LIN {X -0.149,Y -605.682,Z 1425.041,A 0.000,B 0.000,C 90.000,E1 43.299} C_DIS
LIN {X -0.289,Y -605.290,Z 1425.036,A 0.000,B 0.000,C 90.000,E1 42.528} C_DIS
LIN {X -0.379,Y -604.390,Z 1425.029,A 0.000,B 0.000,C 90.000,E1 41.229} C_DIS
LIN {X -0.024,Y -603.135,Z 1425.022,A 0.000,B 0.000,C 90.000,E1 39.886} C_DIS
LIN {X -0.162,Y -601.577,Z 1425.014,A 0.000,B 0.000,C 90.000,E1 38.588} C_DIS
LIN {X 0.234,Y -599.735,Z 1425.007,A 0.000,B 0.000,C 90.000,E1 37.237} C_DIS
LIN {X 0.126,Y -598.447,Z 1425.003,A 0.000,B 0.000,C 90.000,E1 36.457} C_DIS
LIN {X 0.240,Y -596.428,Z 1424.997,A 0.000,B 0.000,C 90.000,E1 35.391} C_DIS
LIN {X 0.320,Y -594.156,Z 1424.991,A 0.000,B 0.000,C 90.000,E1 34.326} C_DIS
LIN {X -0.182,Y -592.218,Z 1424.986,A 0.000,B 0.000,C 90.000,E1 33.579} C_DIS
LIN {X 0.002,Y -589.416,Z 1424.981,A 0.000,B 0.000,C 90.000,E1 32.498} C_DIS
LIN {X 0.081,Y -587.834,Z 1424.978,A 0.000,B 0.000,C 90.000,E1 31.957} C_DIS
LIN {X 0.202,Y -584.213,Z 1424.972,A 0.000,B 0.000,C 90.000,E1 30.875} C_DIS
LIN {X 0.242,Y -582.162,Z 1424.969,A 0.000,B 0.000,C 90.000,E1 30.335} C_DIS
LIN {X 0.125,Y -578.746,Z 1424.964,A 0.000,B 0.000,C 90.000,E1 29.539} C_DIS
LIN {X 0.044,Y -575.611,Z 1424.960,A 0.000,B 0.000,C 90.000,E1 28.871} C_DIS
LIN {X 0.083,Y -571.423,Z 1424.956,A 0.000,B 0.000,C 90.000,E1 28.052} C_DIS
LIN {X -0.156,Y -566.922,Z 1424.951,A 0.000,B 0.000,C 90.000,E1 27.257} C_DIS
LIN {X 0.149,Y -562.893,Z 1424.948,A 0.000,B 0.000,C 90.000,E1 26.539} C_DIS
LIN {X 0.164,Y -558.566,Z 1424.944,A 0.000,B 0.000,C 90.000,E1 25.848} C_DIS
LIN {X -0.249,Y -554.890,Z 1424.941,A 0.000,B 0.000,C 90.000,E1 25.335} C_DIS
LIN {X 0.087,Y -549.144,Z 1424.936,A 0.000,B 0.000,C 90.000,E1 24.463} C_DIS
LIN {X -0.139,Y -542.747,Z 1424.931,A 0.000,B 0.000,C 90.000,E1 23.643} C_DIS
LIN {X 0.201,Y -536.969,Z 1424.927,A 0.000,B 0.000,C 90.000,E1 22.898} C_DIS
LIN {X 0.031,Y -526.966,Z 1424.921,A 0.000,B 0.000,C 90.000,E1 21.770} C_DIS
LIN {X 0.093,Y -518.065,Z 1424.916,A 0.000,B 0.000,C 90.000,E1 20.791} C_DIS
LIN {X 0.008,Y -507.294,Z 1424.909,A 0.000,B 0.000,C 90.000,E1 19.685} C_DIS
LIN {X 0.004,Y -496.701,Z 1424.903,A 0.000,B 0.000,C 90.000,E1 18.598} C_DIS
LIN {X 0.166,Y -481.870,Z 1424.895,A 0.000,B 0.000,C 90.000,E1 17.040} C_DIS
LIN {X -0.202,Y -472.414,Z 1424.889,A 0.000,B 0.000,C 90.000,E1 16.079} C_DIS
LIN {X 0.092,Y -458.896,Z 1424.881,A 0.000,B 0.000,C 90.000,E1 14.537} C_DIS
LIN {X 0.134,Y -445.461,Z 1424.872,A 0.000,B 0.000,C 90.000,E1 13.008} C_DIS
LIN {X 0.001,Y -434.836,Z 1424.865,A 0.000,B 0.000,C 90.000,E1 11.771} C_DIS
LIN {X 0.035,Y -418.788,Z 1424.854,A 0.000,B 0.000,C 90.000,E1 9.792} C_DIS
LIN {X -0.090,Y -411.731,Z 1424.850,A 0.000,B 0.000,C 90.000,E1 8.973} C_DIS
LIN {X -0.154,Y -405.705,Z 1424.846,A 0.000,B 0.000,C 90.000,E1 8.341} C_DIS
LIN {X 0.152,Y -402.589,Z 1424.845,A 0.000,B 0.000,C 90.000,E1 7.992} C_DIS
LIN {X 0.137,Y -399.167,Z 1424.843,A 0.000,B 0.000,C 90.000,E1 7.701} C_DIS
LIN {X -0.075,Y -395.542,Z 1424.841,A 0.000,B 0.000,C 90.000,E1 7.466} C_DIS
LIN {X -0.184,Y -393.227,Z 1424.841,A 0.000,B 0.000,C 90.000,E1 7.352} C_DIS
LIN {X 0.009,Y -390.894,Z 1424.840,A 0.000,B 0.000,C 90.000,E1 7.239} C_DIS
LIN {X -0.074,Y -390.220,Z 1424.840,A 0.000,B 0.000,C 90.000,E1 7.239} C_DIS
LIN {X -0.094,Y -363.864,Z 1424.840,A 0.000,B 0.000,C 90.000,E1 7.239} C_DIS
LIN {X 0.000,Y -360.905,Z 1424.802,A 0.000,B 0.000,C 90.000,E1 0.286} C_DIS
LIN {X -0.053,Y -359.426,Z 1424.770,A 0.000,B 0.000,C 90.000,E1 354.546} C_DIS
LIN {X 0.070,Y -358.890,Z 1424.759,A 0.000,B 0.000,C 90.000,E1 352.648} C_DIS
LIN {X -0.020,Y -359.563,Z 1424.726,A 0.000,B 0.000,C 90.000,E1 346.645} C_DIS
LIN {X 0.001,Y -361.801,Z 1424.684,A 0.000,B 0.000,C 90.000,E1 339.135} C_DIS
LIN {X -0.154,Y -362.053,Z 1424.680,A 0.000,B 0.000,C 90.000,E1 338.411} C_DIS
LIN {X 0.189,Y -365.980,Z 1424.643,A 0.000,B 0.000,C 90.000,E1 331.641} C_DIS
LIN {X 0.029,Y -366.387,Z 1424.639,A 0.000,B 0.000,C 90.000,E1 330.923} C_DIS
LIN {X -0.031,Y -371.355,Z 1424.604,A 0.000,B 0.000,C 90.000,E1 324.642} C_DIS
LIN {X -0.043,Y -371.766,Z 1424.602,A 0.000,B 0.000,C 90.000,E1 324.276} C_DIS
LIN {X 0.013,Y -377.358,Z 1424.567,A 0.000,B 0.000,C 90.000,E1 318.038} C_DIS
LIN {X 0.012,Y -378.235,Z 1424.563,A 0.000,B 0.000,C 90.000,E1 317.310} C_DIS
LIN {X 0.002,Y -383.940,Z 1424.531,A 0.000,B 0.000,C 90.000,E1 311.515} C_DIS
LIN {X 0.088,Y -384.893,Z 1424.527,A 0.000,B 0.000,C 90.000,E1 310.782} C_DIS
LIN {X 0.262,Y -390.610,Z 1424.495,A 0.000,B 0.000,C 90.000,E1 305.025} C_DIS
LIN {X 0.106,Y -391.104,Z 1424.493,A 0.000,B 0.000,C 90.000,E1 304.692} C_DIS
LIN {X 0.022,Y -391.648,Z 1424.489,A 0.000,B 0.000,C 90.000,E1 303.992} C_DIS
LIN {X -0.080,Y -396.825,Z 1424.459,A 0.000,B 0.000,C 90.000,E1 298.693} C_DIS
LIN {X -0.210,Y -397.120,Z 1424.457,A 0.000,B 0.000,C 90.000,E1 298.359} C_DIS
LIN {X -0.055,Y -401.597,Z 1424.426,A 0.000,B 0.000,C 90.000,E1 292.717} C_DIS
LIN {X 0.222,Y -404.659,Z 1424.395,A 0.000,B 0.000,C 90.000,E1 287.094} C_DIS
LIN {X -0.079,Y -404.735,Z 1424.391,A 0.000,B 0.000,C 90.000,E1 286.441} C_DIS
LIN {X 0.214,Y -406.099,Z 1424.364,A 0.000,B 0.000,C 90.000,E1 281.535} C_DIS
LIN {X -0.176,Y -406.094,Z 1424.362,A 0.000,B 0.000,C 90.000,E1 281.243} C_DIS
LIN {X -0.097,Y -405.680,Z 1424.333,A 0.000,B 0.000,C 90.000,E1 276.024} C_DIS
LIN {X -0.165,Y -405.058,Z 1424.328,A 0.000,B 0.000,C 90.000,E1 274.992} C_DIS
LIN {X -0.060,Y -403.497,Z 1424.304,A 0.000,B 0.000,C 90.000,E1 270.802} C_DIS
LIN {X -0.092,Y -403.288,Z 1424.302,A 0.000,B 0.000,C 90.000,E1 270.458} C_DIS
LIN {X 0.091,Y -398.931,Z 1424.271,A 0.000,B 0.000,C 90.000,E1 264.837} C_DIS
LIN {X -0.040,Y -393.108,Z 1424.242,A 0.000,B 0.000,C 90.000,E1 259.567} C_DIS
LIN {X -0.079,Y -392.835,Z 1424.240,A 0.000,B 0.000,C 90.000,E1 259.218} C_DIS
LIN {X 0.034,Y -385.993,Z 1424.212,A 0.000,B 0.000,C 90.000,E1 254.212} C_DIS
LIN {X -0.026,Y -385.267,Z 1424.208,A 0.000,B 0.000,C 90.000,E1 253.504} C_DIS
LIN {X -0.004,Y -384.768,Z 1424.206,A 0.000,B 0.000,C 90.000,E1 253.142} C_DIS
LIN {X 0.221,Y -377.973,Z 1424.182,A 0.000,B 0.000,C 90.000,E1 248.773} C_DIS
LIN {X -0.044,Y -376.233,Z 1424.174,A 0.000,B 0.000,C 90.000,E1 247.358} C_DIS
LIN {X 0.057,Y -374.944,Z 1424.170,A 0.000,B 0.000,C 90.000,E1 246.613} C_DIS
LIN {X -0.208,Y -368.417,Z 1424.148,A 0.000,B 0.000,C 90.000,E1 242.615} C_DIS
LIN {X 0.097,Y -366.047,Z 1424.137,A 0.000,B 0.000,C 90.000,E1 240.717} C_DIS
LIN {X 0.004,Y -359.196,Z 1424.115,A 0.000,B 0.000,C 90.000,E1 236.628} C_DIS
LIN {X 0.021,Y -355.842,Z 1424.100,A 0.000,B 0.000,C 90.000,E1 233.989} C_DIS
LIN {X -0.173,Y -348.793,Z 1424.075,A 0.000,B 0.000,C 90.000,E1 229.461} C_DIS
LIN {X -0.097,Y -346.185,Z 1424.062,A 0.000,B 0.000,C 90.000,E1 227.148} C_DIS
LIN {X -0.088,Y -345.065,Z 1424.058,A 0.000,B 0.000,C 90.000,E1 226.377} C_DIS
LIN {X 0.094,Y -338.586,Z 1424.030,A 0.000,B 0.000,C 90.000,E1 221.310} C_DIS
LIN {X 0.094,Y -336.840,Z 1424.019,A 0.000,B 0.000,C 90.000,E1 219.358} C_DIS
LIN {X 0.014,Y -330.861,Z 1423.988,A 0.000,B 0.000,C 90.000,E1 213.865} C_DIS
LIN {X 0.149,Y -329.296,Z 1423.975,A 0.000,B 0.000,C 90.000,E1 211.465} C_DIS
LIN {X -0.154,Y -324.669,Z 1423.942,A 0.000,B 0.000,C 90.000,E1 205.540} C_DIS
LIN {X 0.174,Y -323.837,Z 1423.928,A 0.000,B 0.000,C 90.000,E1 203.078} C_DIS
LIN {X -0.017,Y -321.124,Z 1423.881,A 0.000,B 0.000,C 90.000,E1 194.662} C_DIS
LIN {X 0.138,Y -320.932,Z 1423.877,A 0.000,B 0.000,C 90.000,E1 193.828} C_DIS
LIN {X -0.076,Y -321.562,Z 1423.832,A 0.000,B 0.000,C 90.000,E1 185.796} C_DIS
LIN {X -0.143,Y -324.415,Z 1423.790,A 0.000,B 0.000,C 90.000,E1 178.165} C_DIS
LIN {X -0.141,Y -325.376,Z 1423.783,A 0.000,B 0.000,C 90.000,E1 176.963} C_DIS
LIN {X -0.063,Y -328.044,Z 1423.757,A 0.000,B 0.000,C 90.000,E1 172.186} C_DIS
LIN {X -0.081,Y -333.268,Z 1423.757,A 0.000,B 0.000,C 90.000,E1 172.186} C_DIS
LIN {X 0.104,Y -333.888,Z 1423.756,A 0.000,B 0.000,C 90.000,E1 172.129} C_DIS
LIN {X -0.027,Y -335.075,Z 1423.756,A 0.000,B 0.000,C 90.000,E1 172.008} C_DIS
LIN {X -0.051,Y -338.203,Z 1423.751,A 0.000,B 0.000,C 90.000,E1 171.254} C_DIS
LIN {X 0.127,Y -343.292,Z 1423.747,A 0.000,B 0.000,C 90.000,E1 170.443} C_DIS
LIN {X -0.064,Y -351.327,Z 1423.741,A 0.000,B 0.000,C 90.000,E1 169.398} C_DIS
LIN {X 0.033,Y -356.948,Z 1423.737,A 0.000,B 0.000,C 90.000,E1 168.634} C_DIS
LIN {X -0.093,Y -371.061,Z 1423.727,A 0.000,B 0.000,C 90.000,E1 166.825} C_DIS
LIN {X 0.020,Y -384.413,Z 1423.718,A 0.000,B 0.000,C 90.000,E1 165.283} C_DIS
LIN {X 0.103,Y -396.641,Z 1423.711,A 0.000,B 0.000,C 90.000,E1 164.031} C_DIS
LIN {X 0.071,Y -415.293,Z 1423.702,A 0.000,B 0.000,C 90.000,E1 162.362} C_DIS
LIN {X -0.097,Y -427.764,Z 1423.696,A 0.000,B 0.000,C 90.000,E1 161.329} C_DIS
LIN {X 0.095,Y -443.406,Z 1423.689,A 0.000,B 0.000,C 90.000,E1 160.007} C_DIS
LIN {X 0.078,Y -457.201,Z 1423.683,A 0.000,B 0.000,C 90.000,E1 158.847} C_DIS
LIN {X -0.139,Y -469.354,Z 1423.677,A 0.000,B 0.000,C 90.000,E1 157.847} C_DIS
LIN {X -0.008,Y -479.683,Z 1423.672,A 0.000,B 0.000,C 90.000,E1 156.922} C_DIS
LIN {X 0.239,Y -488.387,Z 1423.667,A 0.000,B 0.000,C 90.000,E1 156.102} C_DIS
LIN {X -0.160,Y -494.067,Z 1423.664,A 0.000,B 0.000,C 90.000,E1 155.613} C_DIS
LIN {X -0.021,Y -499.605,Z 1423.661,A 0.000,B 0.000,C 90.000,E1 155.049} C_DIS
LIN {X 0.098,Y -506.416,Z 1423.657,A 0.000,B 0.000,C 90.000,E1 154.332} C_DIS
LIN {X -0.140,Y -512.807,Z 1423.654,A 0.000,B 0.000,C 90.000,E1 153.640} C_DIS
LIN {X -0.124,Y -517.609,Z 1423.650,A 0.000,B 0.000,C 90.000,E1 153.050} C_DIS
LIN {X 0.252,Y -522.911,Z 1423.646,A 0.000,B 0.000,C 90.000,E1 152.281} C_DIS
LIN {X -0.070,Y -524.998,Z 1423.645,A 0.000,B 0.000,C 90.000,E1 152.025} C_DIS
LIN {X -0.137,Y -529.380,Z 1423.641,A 0.000,B 0.000,C 90.000,E1 151.307} C_DIS
LIN {X -0.018,Y -532.581,Z 1423.637,A 0.000,B 0.000,C 90.000,E1 150.717} C_DIS
LIN {X -0.019,Y -535.956,Z 1423.633,A 0.000,B 0.000,C 90.000,E1 149.999} C_DIS
LIN {X 0.148,Y -538.361,Z 1423.630,A 0.000,B 0.000,C 90.000,E1 149.410} C_DIS
LIN {X -0.133,Y -540.566,Z 1423.627,A 0.000,B 0.000,C 90.000,E1 148.869} C_DIS
LIN {X 0.074,Y -543.361,Z 1423.622,A 0.000,B 0.000,C 90.000,E1 147.995} C_DIS
LIN {X -0.146,Y -545.849,Z 1423.618,A 0.000,B 0.000,C 90.000,E1 147.168} C_DIS
LIN {X 0.345,Y -546.656,Z 1423.616,A 0.000,B 0.000,C 90.000,E1 146.834} C_DIS
LIN {X -0.053,Y -549.998,Z 1423.608,A 0.000,B 0.000,C 90.000,E1 145.468} C_DIS
LIN {X 0.171,Y -552.114,Z 1423.602,A 0.000,B 0.000,C 90.000,E1 144.322} C_DIS
LIN {X -0.090,Y -552.630,Z 1423.600,A 0.000,B 0.000,C 90.000,E1 144.069} C_DIS
LIN {X 0.173,Y -554.065,Z 1423.594,A 0.000,B 0.000,C 90.000,E1 142.924} C_DIS
LIN {X 0.019,Y -555.361,Z 1423.588,A 0.000,B 0.000,C 90.000,E1 141.823} C_DIS
LIN {X 0.038,Y -556.891,Z 1423.579,A 0.000,B 0.000,C 90.000,E1 140.150} C_DIS
LIN {X 0.202,Y -557.572,Z 1423.574,A 0.000,B 0.000,C 90.000,E1 139.299} C_DIS
LIN {X 0.119,Y -558.510,Z 1423.566,A 0.000,B 0.000,C 90.000,E1 137.919} C_DIS
LIN {X 0.045,Y -559.293,Z 1423.559,A 0.000,B 0.000,C 90.000,E1 136.539} C_DIS
LIN {X -0.037,Y -559.970,Z 1423.551,A 0.000,B 0.000,C 90.000,E1 135.162} C_DIS
LIN {X -0.238,Y -560.255,Z 1423.546,A 0.000,B 0.000,C 90.000,E1 134.352} C_DIS
LIN {X -0.230,Y -560.689,Z 1423.537,A 0.000,B 0.000,C 90.000,E1 132.690} C_DIS
LIN {X 0.068,Y -560.743,Z 1423.531,A 0.000,B 0.000,C 90.000,E1 131.553} C_DIS
LIN {X 0.129,Y -560.895,Z 1423.522,A 0.000,B 0.000,C 90.000,E1 129.886} C_DIS
LIN {X -0.265,Y -560.978,Z 1423.514,A 0.000,B 0.000,C 90.000,E1 128.543} C_DIS
LIN {X -0.225,Y -561.036,Z 1423.506,A 0.000,B 0.000,C 90.000,E1 127.156} C_DIS
LIN {X 0.259,Y -560.967,Z 1423.499,A 0.000,B 0.000,C 90.000,E1 125.724} C_DIS
LIN {X 0.093,Y -560.896,Z 1423.491,A 0.000,B 0.000,C 90.000,E1 124.358} C_DIS
LIN {X 0.247,Y -560.680,Z 1423.483,A 0.000,B 0.000,C 90.000,E1 122.959} C_DIS
LIN {X -0.220,Y -561.187,Z 1423.456,A 0.000,B 0.000,C 90.000,E1 118.025} C_DIS
LIN {X -0.158,Y -561.922,Z 1423.446,A 0.000,B 0.000,C 90.000,E1 116.360} C_DIS
LIN {X -0.241,Y -562.267,Z 1423.442,A 0.000,B 0.000,C 90.000,E1 115.540} C_DIS
LIN {X -0.270,Y -562.870,Z 1423.430,A 0.000,B 0.000,C 90.000,E1 113.334} C_DIS
LIN {X -0.148,Y -563.337,Z 1423.427,A 0.000,B 0.000,C 90.000,E1 112.770} C_DIS
LIN {X 0.075,Y -564.151,Z 1423.424,A 0.000,B 0.000,C 90.000,E1 112.333} C_DIS
LIN {X -0.296,Y -564.870,Z 1423.423,A 0.000,B 0.000,C 90.000,E1 112.153} C_DIS
LIN {X 0.150,Y -567.341,Z 1423.421,A 0.000,B 0.000,C 90.000,E1 111.770} C_DIS
LIN {X -0.062,Y -570.457,Z 1423.420,A 0.000,B 0.000,C 90.000,E1 111.589} C_DIS
LIN {X 0.224,Y -572.267,Z 1423.419,A 0.000,B 0.000,C 90.000,E1 111.461} C_DIS
LIN {X -0.331,Y -578.293,Z 1423.418,A 0.000,B 0.000,C 90.000,E1 111.227} C_DIS
LIN {X -0.141,Y -581.400,Z 1423.417,A 0.000,B 0.000,C 90.000,E1 111.046} C_DIS
LIN {X 0.121,Y -587.184,Z 1423.415,A 0.000,B 0.000,C 90.000,E1 110.663} C_DIS
LIN {X 0.193,Y -592.703,Z 1423.413,A 0.000,B 0.000,C 90.000,E1 110.248} C_DIS
LIN {X -0.209,Y -595.303,Z 1423.411,A 0.000,B 0.000,C 90.000,E1 110.066} C_DIS
LIN {X -0.160,Y -600.564,Z 1423.409,A 0.000,B 0.000,C 90.000,E1 109.577} C_DIS
LIN {X -0.266,Y -604.414,Z 1423.407,A 0.000,B 0.000,C 90.000,E1 109.214} C_DIS
LIN {X 0.013,Y -610.350,Z 1423.403,A 0.000,B 0.000,C 90.000,E1 108.544} C_DIS
LIN {X -0.282,Y -613.705,Z 1423.401,A 0.000,B 0.000,C 90.000,E1 108.181} C_DIS
LIN {X -0.030,Y -618.411,Z 1423.397,A 0.000,B 0.000,C 90.000,E1 107.511} C_DIS
LIN {X 0.055,Y -623.124,Z 1423.393,A 0.000,B 0.000,C 90.000,E1 106.732} C_DIS
LIN {X 0.010,Y -626.256,Z 1423.389,A 0.000,B 0.000,C 90.000,E1 105.969} C_DIS
LIN {X -0.233,Y -627.634,Z 1423.386,A 0.000,B 0.000,C 90.000,E1 105.481} C_DIS
LIN {X -0.226,Y -629.141,Z 1423.382,A 0.000,B 0.000,C 90.000,E1 104.717} C_DIS
LIN {X 0.181,Y -630.839,Z 1423.375,A 0.000,B 0.000,C 90.000,E1 103.411} C_DIS
LIN {X -0.202,Y -631.423,Z 1423.372,A 0.000,B 0.000,C 90.000,E1 102.939} C_DIS
LIN {X -0.155,Y -631.557,Z 1423.368,A 0.000,B 0.000,C 90.000,E1 102.175} C_DIS
LIN {X -0.045,Y -631.402,Z 1423.365,A 0.000,B 0.000,C 90.000,E1 101.658} C_DIS
LIN {X 0.194,Y -630.971,Z 1423.362,A 0.000,B 0.000,C 90.000,E1 101.130} C_DIS
LIN {X -0.191,Y -630.309,Z 1423.359,A 0.000,B 0.000,C 90.000,E1 100.658} C_DIS
LIN {X -0.273,Y -628.857,Z 1423.355,A 0.000,B 0.000,C 90.000,E1 99.905} C_DIS
LIN {X -0.058,Y -627.605,Z 1423.352,A 0.000,B 0.000,C 90.000,E1 99.378} C_DIS
LIN {X -0.166,Y -625.145,Z 1423.348,A 0.000,B 0.000,C 90.000,E1 98.624} C_DIS
LIN {X 0.144,Y -624.276,Z 1423.346,A 0.000,B 0.000,C 90.000,E1 98.341} C_DIS
LIN {X 0.318,Y -622.179,Z 1423.344,A 0.000,B 0.000,C 90.000,E1 97.814} C_DIS
LIN {X -0.224,Y -619.751,Z 1423.341,A 0.000,B 0.000,C 90.000,E1 97.352} C_DIS
LIN {X 0.123,Y -615.767,Z 1423.337,A 0.000,B 0.000,C 90.000,E1 96.549} C_DIS
LIN {X 0.153,Y -612.884,Z 1423.334,A 0.000,B 0.000,C 90.000,E1 96.030} C_DIS
LIN {X 0.052,Y -608.649,Z 1423.330,A 0.000,B 0.000,C 90.000,E1 95.391} C_DIS
LIN {X -0.025,Y -604.639,Z 1423.327,A 0.000,B 0.000,C 90.000,E1 94.878} C_DIS
LIN {X -0.221,Y -598.405,Z 1423.323,A 0.000,B 0.000,C 90.000,E1 94.245} C_DIS
LIN {X -0.032,Y -591.511,Z 1423.320,A 0.000,B 0.000,C 90.000,E1 93.612} C_DIS
LIN {X -0.022,Y -584.167,Z 1423.317,A 0.000,B 0.000,C 90.000,E1 93.037} C_DIS
LIN {X -0.147,Y -577.666,Z 1423.315,A 0.000,B 0.000,C 90.000,E1 92.636} C_DIS
LIN {X 0.266,Y -573.327,Z 1423.313,A 0.000,B 0.000,C 90.000,E1 92.236} C_DIS
LIN {X 0.229,Y -573.300,Z 1423.313,A 0.000,B 0.000,C 90.000,E1 92.236} C_DIS
LIN {X 0.258,Y -572.433,Z 1423.311,A 0.000,B 0.000,C 90.000,E1 92.007} C_DIS
LIN {X -0.028,Y -572.085,Z 1423.310,A 0.000,B 0.000,C 90.000,E1 91.776} C_DIS
LIN {X 0.269,Y -572.111,Z 1423.307,A 0.000,B 0.000,C 90.000,E1 91.146} C_DIS
LIN {X 0.102,Y -573.642,Z 1423.296,A 0.000,B 0.000,C 90.000,E1 89.255} C_DIS
LIN {X 0.119,Y -574.706,Z 1423.290,A 0.000,B 0.000,C 90.000,E1 88.165} C_DIS
LIN {X -0.120,Y -576.210,Z 1423.281,A 0.000,B 0.000,C 90.000,E1 86.560} C_DIS
LIN {X 0.130,Y -577.521,Z 1423.273,A 0.000,B 0.000,C 90.000,E1 85.179} C_DIS
LIN {X -0.029,Y -579.110,Z 1423.264,A 0.000,B 0.000,C 90.000,E1 83.571} C_DIS
LIN {X 0.197,Y -581.218,Z 1423.254,A 0.000,B 0.000,C 90.000,E1 81.659} C_DIS
LIN {X 0.012,Y -582.669,Z 1423.246,A 0.000,B 0.000,C 90.000,E1 80.330} C_DIS
LIN {X -0.061,Y -584.115,Z 1423.239,A 0.000,B 0.000,C 90.000,E1 78.993} C_DIS
LIN {X 0.003,Y -585.507,Z 1423.231,A 0.000,B 0.000,C 90.000,E1 77.645} C_DIS
LIN {X -0.156,Y -586.366,Z 1423.225,A 0.000,B 0.000,C 90.000,E1 76.589} C_DIS
LIN {X 0.084,Y -587.323,Z 1423.218,A 0.000,B 0.000,C 90.000,E1 75.227} C_DIS
LIN {X -0.225,Y -588.223,Z 1423.211,A 0.000,B 0.000,C 90.000,E1 73.921} C_DIS
LIN {X 0.309,Y -589.296,Z 1423.200,A 0.000,B 0.000,C 90.000,E1 72.000} C_DIS
LIN {X 0.070,Y -590.121,Z 1423.191,A 0.000,B 0.000,C 90.000,E1 70.423} C_DIS
LIN {X -0.159,Y -590.992,Z 1423.182,A 0.000,B 0.000,C 90.000,E1 68.847} C_DIS
LIN {X 0.054,Y -591.465,Z 1423.178,A 0.000,B 0.000,C 90.000,E1 68.028} C_DIS
LIN {X -0.050,Y -592.677,Z 1423.168,A 0.000,B 0.000,C 90.000,E1 66.177} C_DIS
LIN {X 0.253,Y -594.107,Z 1423.156,A 0.000,B 0.000,C 90.000,E1 64.024} C_DIS
LIN {X -0.203,Y -595.211,Z 1423.149,A 0.000,B 0.000,C 90.000,E1 62.743} C_DIS
LIN {X 0.070,Y -596.501,Z 1423.140,A 0.000,B 0.000,C 90.000,E1 61.129} C_DIS
LIN {X 0.049,Y -598.081,Z 1423.129,A 0.000,B 0.000,C 90.000,E1 59.282} C_DIS
LIN {X -0.048,Y -599.595,Z 1423.121,A 0.000,B 0.000,C 90.000,E1 57.709} C_DIS
LIN {X -0.102,Y -601.023,Z 1423.112,A 0.000,B 0.000,C 90.000,E1 56.135} C_DIS
LIN {X -0.041,Y -602.230,Z 1423.105,A 0.000,B 0.000,C 90.000,E1 54.815} C_DIS
LIN {X -0.196,Y -603.473,Z 1423.096,A 0.000,B 0.000,C 90.000,E1 53.256} C_DIS
LIN {X 0.251,Y -604.448,Z 1423.089,A 0.000,B 0.000,C 90.000,E1 51.904} C_DIS
LIN {X -0.238,Y -605.378,Z 1423.081,A 0.000,B 0.000,C 90.000,E1 50.642} C_DIS
LIN {X 0.141,Y -605.972,Z 1423.074,A 0.000,B 0.000,C 90.000,E1 49.299} C_DIS
LIN {X 0.264,Y -606.187,Z 1423.068,A 0.000,B 0.000,C 90.000,E1 48.243} C_DIS
LIN {X -0.389,Y -606.415,Z 1423.057,A 0.000,B 0.000,C 90.000,E1 46.215} C_DIS
LIN {X -0.104,Y -606.397,Z 1423.052,A 0.000,B 0.000,C 90.000,E1 45.405} C_DIS
LIN {X -0.007,Y -606.276,Z 1423.046,A 0.000,B 0.000,C 90.000,E1 44.352} C_DIS
LIN {X -0.112,Y -605.689,Z 1423.039,A 0.000,B 0.000,C 90.000,E1 43.056} C_DIS
LIN {X -0.001,Y -605.092,Z 1423.033,A 0.000,B 0.000,C 90.000,E1 42.000} C_DIS
LIN {X -0.144,Y -604.541,Z 1423.029,A 0.000,B 0.000,C 90.000,E1 41.229} C_DIS
LIN {X 0.003,Y -603.016,Z 1423.020,A 0.000,B 0.000,C 90.000,E1 39.644} C_DIS
LIN {X -0.047,Y -601.434,Z 1423.013,A 0.000,B 0.000,C 90.000,E1 38.338} C_DIS
LIN {X -0.120,Y -599.561,Z 1423.006,A 0.000,B 0.000,C 90.000,E1 37.030} C_DIS
LIN {X 0.013,Y -597.718,Z 1423.000,A 0.000,B 0.000,C 90.000,E1 35.964} C_DIS
LIN {X -0.113,Y -596.146,Z 1422.995,A 0.000,B 0.000,C 90.000,E1 35.185} C_DIS
LIN {X -0.036,Y -593.802,Z 1422.990,A 0.000,B 0.000,C 90.000,E1 34.119} C_DIS
LIN {X 0.280,Y -591.818,Z 1422.985,A 0.000,B 0.000,C 90.000,E1 33.293} C_DIS
LIN {X -0.242,Y -589.736,Z 1422.981,A 0.000,B 0.000,C 90.000,E1 32.546} C_DIS
LIN {X 0.025,Y -587.266,Z 1422.976,A 0.000,B 0.000,C 90.000,E1 31.720} C_DIS
LIN {X -0.168,Y -583.634,Z 1422.970,A 0.000,B 0.000,C 90.000,E1 30.669} C_DIS
LIN {X -0.133,Y -581.498,Z 1422.967,A 0.000,B 0.000,C 90.000,E1 30.129} C_DIS
LIN {X 0.247,Y -577.924,Z 1422.963,A 0.000,B 0.000,C 90.000,E1 29.283} C_DIS
LIN {X 0.235,Y -575.366,Z 1422.960,A 0.000,B 0.000,C 90.000,E1 28.743} C_DIS
LIN {X -0.154,Y -571.875,Z 1422.956,A 0.000,B 0.000,C 90.000,E1 28.103} C_DIS
LIN {X 0.115,Y -567.415,Z 1422.952,A 0.000,B 0.000,C 90.000,E1 27.257} C_DIS
LIN {X 0.171,Y -563.420,Z 1422.948,A 0.000,B 0.000,C 90.000,E1 26.565} C_DIS
LIN {X -0.063,Y -559.110,Z 1422.944,A 0.000,B 0.000,C 90.000,E1 25.899} C_DIS
LIN {X 0.028,Y -555.475,Z 1422.941,A 0.000,B 0.000,C 90.000,E1 25.335} C_DIS
LIN {X -0.132,Y -549.755,Z 1422.936,A 0.000,B 0.000,C 90.000,E1 24.515} C_DIS
LIN {X -0.227,Y -544.447,Z 1422.932,A 0.000,B 0.000,C 90.000,E1 23.823} C_DIS
LIN {X 0.259,Y -539.973,Z 1422.929,A 0.000,B 0.000,C 90.000,E1 23.206} C_DIS
LIN {X 0.214,Y -535.149,Z 1422.926,A 0.000,B 0.000,C 90.000,E1 22.642} C_DIS
LIN {X -0.210,Y -527.877,Z 1422.921,A 0.000,B 0.000,C 90.000,E1 21.844} C_DIS
LIN {X 0.201,Y -517.406,Z 1422.915,A 0.000,B 0.000,C 90.000,E1 20.663} C_DIS
LIN {X -0.086,Y -506.584,Z 1422.909,A 0.000,B 0.000,C 90.000,E1 19.577} C_DIS
LIN {X -0.039,Y -497.110,Z 1422.903,A 0.000,B 0.000,C 90.000,E1 18.598} C_DIS
LIN {X 0.148,Y -481.091,Z 1422.894,A 0.000,B 0.000,C 90.000,E1 16.913} C_DIS
LIN {X -0.188,Y -463.633,Z 1422.884,A 0.000,B 0.000,C 90.000,E1 15.064} C_DIS
LIN {X -0.108,Y -454.342,Z 1422.878,A 0.000,B 0.000,C 90.000,E1 14.008} C_DIS
LIN {X 0.105,Y -436.741,Z 1422.867,A 0.000,B 0.000,C 90.000,E1 11.951} C_DIS
LIN {X 0.103,Y -418.131,Z 1422.854,A 0.000,B 0.000,C 90.000,E1 9.670} C_DIS
LIN {X -0.175,Y -411.542,Z 1422.849,A 0.000,B 0.000,C 90.000,E1 8.859} C_DIS
LIN {X -0.018,Y -404.426,Z 1422.844,A 0.000,B 0.000,C 90.000,E1 7.992} C_DIS
LIN {X -0.183,Y -399.847,Z 1422.842,A 0.000,B 0.000,C 90.000,E1 7.530} C_DIS
LIN {X -0.153,Y -394.986,Z 1422.839,A 0.000,B 0.000,C 90.000,E1 7.068} C_DIS
LIN {X -0.069,Y -391.494,Z 1422.838,A 0.000,B 0.000,C 90.000,E1 6.777} C_DIS
LIN {X 0.199,Y -387.722,Z 1422.836,A 0.000,B 0.000,C 90.000,E1 6.486} C_DIS
LIN {X -0.053,Y -385.738,Z 1422.836,A 0.000,B 0.000,C 90.000,E1 6.429} C_DIS
LIN {X 0.021,Y -383.960,Z 1422.835,A 0.000,B 0.000,C 90.000,E1 6.372} C_DIS
LIN {X -0.010,Y -363.201,Z 1422.835,A 0.000,B 0.000,C 90.000,E1 6.372} C_DIS
LIN {X -0.158,Y -360.906,Z 1422.802,A 0.000,B 0.000,C 90.000,E1 0.344} C_DIS
LIN {X -0.029,Y -359.468,Z 1422.778,A 0.000,B 0.000,C 90.000,E1 356.045} C_DIS
LIN {X -0.053,Y -359.426,Z 1422.770,A 0.000,B 0.000,C 90.000,E1 354.546} C_DIS
LIN {X 0.070,Y -358.890,Z 1422.759,A 0.000,B 0.000,C 90.000,E1 352.648} C_DIS
LIN {X -0.020,Y -359.563,Z 1422.726,A 0.000,B 0.000,C 90.000,E1 346.645} C_DIS
LIN {X 0.001,Y -361.801,Z 1422.684,A 0.000,B 0.000,C 90.000,E1 339.135} C_DIS
LIN {X -0.154,Y -362.053,Z 1422.680,A 0.000,B 0.000,C 90.000,E1 338.411} C_DIS
LIN {X 0.189,Y -365.980,Z 1422.643,A 0.000,B 0.000,C 90.000,E1 331.641} C_DIS
LIN {X 0.029,Y -366.387,Z 1422.639,A 0.000,B 0.000,C 90.000,E1 330.923} C_DIS
LIN {X -0.031,Y -371.355,Z 1422.604,A 0.000,B 0.000,C 90.000,E1 324.642} C_DIS
LIN {X -0.043,Y -371.766,Z 1422.602,A 0.000,B 0.000,C 90.000,E1 324.276} C_DIS
LIN {X 0.013,Y -377.358,Z 1422.567,A 0.000,B 0.000,C 90.000,E1 318.038} C_DIS
LIN {X 0.012,Y -378.235,Z 1422.563,A 0.000,B 0.000,C 90.000,E1 317.310} C_DIS
LIN {X 0.002,Y -383.940,Z 1422.531,A 0.000,B 0.000,C 90.000,E1 311.515} C_DIS
LIN {X 0.088,Y -384.893,Z 1422.527,A 0.000,B 0.000,C 90.000,E1 310.782} C_DIS
LIN {X 0.262,Y -390.610,Z 1422.495,A 0.000,B 0.000,C 90.000,E1 305.025} C_DIS
LIN {X 0.106,Y -391.104,Z 1422.493,A 0.000,B 0.000,C 90.000,E1 304.692} C_DIS
LIN {X 0.022,Y -391.648,Z 1422.489,A 0.000,B 0.000,C 90.000,E1 303.992} C_DIS
LIN {X -0.080,Y -396.825,Z 1422.459,A 0.000,B 0.000,C 90.000,E1 298.693} C_DIS
LIN {X -0.210,Y -397.120,Z 1422.457,A 0.000,B 0.000,C 90.000,E1 298.359} C_DIS
LIN {X -0.055,Y -401.597,Z 1422.426,A 0.000,B 0.000,C 90.000,E1 292.717} C_DIS
LIN {X 0.222,Y -404.659,Z 1422.395,A 0.000,B 0.000,C 90.000,E1 287.094} C_DIS
LIN {X -0.079,Y -404.735,Z 1422.391,A 0.000,B 0.000,C 90.000,E1 286.441} C_DIS
LIN {X 0.214,Y -406.099,Z 1422.364,A 0.000,B 0.000,C 90.000,E1 281.535} C_DIS
LIN {X -0.176,Y -406.094,Z 1422.362,A 0.000,B 0.000,C 90.000,E1 281.243} C_DIS
LIN {X -0.097,Y -405.680,Z 1422.333,A 0.000,B 0.000,C 90.000,E1 276.024} C_DIS
LIN {X -0.165,Y -405.058,Z 1422.328,A 0.000,B 0.000,C 90.000,E1 274.992} C_DIS
LIN {X -0.060,Y -403.497,Z 1422.304,A 0.000,B 0.000,C 90.000,E1 270.802} C_DIS
LIN {X -0.092,Y -403.288,Z 1422.302,A 0.000,B 0.000,C 90.000,E1 270.458} C_DIS
LIN {X 0.091,Y -398.931,Z 1422.271,A 0.000,B 0.000,C 90.000,E1 264.837} C_DIS
LIN {X -0.040,Y -393.108,Z 1422.242,A 0.000,B 0.000,C 90.000,E1 259.567} C_DIS
LIN {X -0.079,Y -392.835,Z 1422.240,A 0.000,B 0.000,C 90.000,E1 259.218} C_DIS
LIN {X 0.034,Y -385.993,Z 1422.212,A 0.000,B 0.000,C 90.000,E1 254.212} C_DIS
LIN {X -0.026,Y -385.267,Z 1422.208,A 0.000,B 0.000,C 90.000,E1 253.504} C_DIS
LIN {X -0.004,Y -384.768,Z 1422.206,A 0.000,B 0.000,C 90.000,E1 253.142} C_DIS
LIN {X 0.221,Y -377.973,Z 1422.182,A 0.000,B 0.000,C 90.000,E1 248.773} C_DIS
LIN {X -0.044,Y -376.233,Z 1422.174,A 0.000,B 0.000,C 90.000,E1 247.358} C_DIS
LIN {X 0.057,Y -374.944,Z 1422.170,A 0.000,B 0.000,C 90.000,E1 246.613} C_DIS
LIN {X -0.208,Y -368.417,Z 1422.148,A 0.000,B 0.000,C 90.000,E1 242.615} C_DIS
LIN {X 0.097,Y -366.047,Z 1422.137,A 0.000,B 0.000,C 90.000,E1 240.717} C_DIS
LIN {X 0.004,Y -359.196,Z 1422.115,A 0.000,B 0.000,C 90.000,E1 236.628} C_DIS
LIN {X 0.021,Y -355.842,Z 1422.100,A 0.000,B 0.000,C 90.000,E1 233.989} C_DIS
LIN {X -0.173,Y -348.793,Z 1422.075,A 0.000,B 0.000,C 90.000,E1 229.461} C_DIS
LIN {X -0.097,Y -346.185,Z 1422.062,A 0.000,B 0.000,C 90.000,E1 227.148} C_DIS
LIN {X -0.088,Y -345.065,Z 1422.058,A 0.000,B 0.000,C 90.000,E1 226.377} C_DIS
LIN {X 0.094,Y -338.586,Z 1422.030,A 0.000,B 0.000,C 90.000,E1 221.310} C_DIS
LIN {X 0.094,Y -336.840,Z 1422.019,A 0.000,B 0.000,C 90.000,E1 219.358} C_DIS
LIN {X 0.014,Y -330.861,Z 1421.988,A 0.000,B 0.000,C 90.000,E1 213.865} C_DIS
LIN {X 0.149,Y -329.296,Z 1421.975,A 0.000,B 0.000,C 90.000,E1 211.465} C_DIS
LIN {X -0.154,Y -324.669,Z 1421.942,A 0.000,B 0.000,C 90.000,E1 205.540} C_DIS
LIN {X 0.174,Y -323.837,Z 1421.928,A 0.000,B 0.000,C 90.000,E1 203.078} C_DIS
LIN {X -0.017,Y -321.124,Z 1421.881,A 0.000,B 0.000,C 90.000,E1 194.662} C_DIS
LIN {X 0.138,Y -320.932,Z 1421.877,A 0.000,B 0.000,C 90.000,E1 193.828} C_DIS
LIN {X -0.076,Y -321.562,Z 1421.832,A 0.000,B 0.000,C 90.000,E1 185.796} C_DIS
LIN {X -0.143,Y -324.415,Z 1421.790,A 0.000,B 0.000,C 90.000,E1 178.165} C_DIS
LIN {X -0.141,Y -325.376,Z 1421.783,A 0.000,B 0.000,C 90.000,E1 176.963} C_DIS
LIN {X 0.068,Y -327.166,Z 1421.763,A 0.000,B 0.000,C 90.000,E1 173.337} C_DIS
LIN {X 0.052,Y -337.143,Z 1421.763,A 0.000,B 0.000,C 90.000,E1 173.337} C_DIS
LIN {X -0.086,Y -338.457,Z 1421.763,A 0.000,B 0.000,C 90.000,E1 173.280} C_DIS
LIN {X -0.102,Y -339.228,Z 1421.761,A 0.000,B 0.000,C 90.000,E1 173.053} C_DIS
LIN {X 0.077,Y -339.480,Z 1421.757,A 0.000,B 0.000,C 90.000,E1 172.243} C_DIS
LIN {X -0.168,Y -339.250,Z 1421.755,A 0.000,B 0.000,C 90.000,E1 171.894} C_DIS
LIN {X 0.071,Y -339.257,Z 1421.754,A 0.000,B 0.000,C 90.000,E1 171.659} C_DIS
LIN {X 0.165,Y -340.160,Z 1421.752,A 0.000,B 0.000,C 90.000,E1 171.254} C_DIS
LIN {X -0.077,Y -340.478,Z 1421.751,A 0.000,B 0.000,C 90.000,E1 171.197} C_DIS
LIN {X -0.009,Y -345.349,Z 1421.746,A 0.000,B 0.000,C 90.000,E1 170.330} C_DIS
LIN {X 0.019,Y -349.923,Z 1421.742,A 0.000,B 0.000,C 90.000,E1 169.634} C_DIS
LIN {X -0.003,Y -363.284,Z 1421.732,A 0.000,B 0.000,C 90.000,E1 167.813} C_DIS
LIN {X -0.057,Y -374.679,Z 1421.724,A 0.000,B 0.000,C 90.000,E1 166.408} C_DIS
LIN {X 0.171,Y -386.610,Z 1421.717,A 0.000,B 0.000,C 90.000,E1 165.046} C_DIS
LIN {X -0.016,Y -398.776,Z 1421.710,A 0.000,B 0.000,C 90.000,E1 163.866} C_DIS
LIN {X 0.121,Y -418.850,Z 1421.701,A 0.000,B 0.000,C 90.000,E1 162.072} C_DIS
LIN {X 0.093,Y -431.242,Z 1421.695,A 0.000,B 0.000,C 90.000,E1 161.040} C_DIS
LIN {X -0.171,Y -445.038,Z 1421.688,A 0.000,B 0.000,C 90.000,E1 159.934} C_DIS
LIN {X -0.198,Y -458.834,Z 1421.682,A 0.000,B 0.000,C 90.000,E1 158.773} C_DIS
LIN {X 0.032,Y -469.477,Z 1421.677,A 0.000,B 0.000,C 90.000,E1 157.847} C_DIS
LIN {X 0.177,Y -479.791,Z 1421.672,A 0.000,B 0.000,C 90.000,E1 156.922} C_DIS
LIN {X -0.213,Y -488.491,Z 1421.668,A 0.000,B 0.000,C 90.000,E1 156.177} C_DIS
LIN {X -0.040,Y -495.552,Z 1421.664,A 0.000,B 0.000,C 90.000,E1 155.485} C_DIS
LIN {X -0.020,Y -502.436,Z 1421.660,A 0.000,B 0.000,C 90.000,E1 154.793} C_DIS
LIN {X -0.039,Y -507.800,Z 1421.657,A 0.000,B 0.000,C 90.000,E1 154.229} C_DIS
LIN {X -0.149,Y -514.117,Z 1421.653,A 0.000,B 0.000,C 90.000,E1 153.512} C_DIS
LIN {X 0.023,Y -517.724,Z 1421.650,A 0.000,B 0.000,C 90.000,E1 153.050} C_DIS
LIN {X 0.112,Y -523.102,Z 1421.646,A 0.000,B 0.000,C 90.000,E1 152.308} C_DIS
LIN {X -0.123,Y -526.062,Z 1421.644,A 0.000,B 0.000,C 90.000,E1 151.897} C_DIS
LIN {X -0.030,Y -529.570,Z 1421.641,A 0.000,B 0.000,C 90.000,E1 151.307} C_DIS
LIN {X 0.092,Y -532.770,Z 1421.637,A 0.000,B 0.000,C 90.000,E1 150.717} C_DIS
LIN {X 0.093,Y -536.143,Z 1421.633,A 0.000,B 0.000,C 90.000,E1 149.999} C_DIS
LIN {X -0.201,Y -538.548,Z 1421.630,A 0.000,B 0.000,C 90.000,E1 149.459} C_DIS
LIN {X -0.018,Y -540.752,Z 1421.627,A 0.000,B 0.000,C 90.000,E1 148.869} C_DIS
LIN {X 0.192,Y -543.546,Z 1421.622,A 0.000,B 0.000,C 90.000,E1 147.995} C_DIS
LIN {X -0.026,Y -546.032,Z 1421.618,A 0.000,B 0.000,C 90.000,E1 147.168} C_DIS
LIN {X -0.255,Y -547.482,Z 1421.615,A 0.000,B 0.000,C 90.000,E1 146.628} C_DIS
LIN {X 0.071,Y -550.119,Z 1421.608,A 0.000,B 0.000,C 90.000,E1 145.468} C_DIS
LIN {X -0.023,Y -552.234,Z 1421.602,A 0.000,B 0.000,C 90.000,E1 144.356} C_DIS
LIN {X 0.101,Y -553.065,Z 1421.599,A 0.000,B 0.000,C 90.000,E1 143.783} C_DIS
LIN {X -0.069,Y -554.454,Z 1421.593,A 0.000,B 0.000,C 90.000,E1 142.683} C_DIS
LIN {X 0.149,Y -555.363,Z 1421.588,A 0.000,B 0.000,C 90.000,E1 141.823} C_DIS
LIN {X 0.169,Y -556.893,Z 1421.579,A 0.000,B 0.000,C 90.000,E1 140.150} C_DIS
LIN {X -0.029,Y -557.575,Z 1421.574,A 0.000,B 0.000,C 90.000,E1 139.337} C_DIS
LIN {X 0.250,Y -558.500,Z 1421.566,A 0.000,B 0.000,C 90.000,E1 137.919} C_DIS
LIN {X -0.159,Y -559.438,Z 1421.557,A 0.000,B 0.000,C 90.000,E1 136.296} C_DIS
LIN {X 0.093,Y -559.928,Z 1421.551,A 0.000,B 0.000,C 90.000,E1 135.162} C_DIS
LIN {X -0.107,Y -560.214,Z 1421.546,A 0.000,B 0.000,C 90.000,E1 134.352} C_DIS
LIN {X -0.101,Y -560.639,Z 1421.537,A 0.000,B 0.000,C 90.000,E1 132.690} C_DIS
LIN {X -0.135,Y -560.689,Z 1421.529,A 0.000,B 0.000,C 90.000,E1 131.310} C_DIS
LIN {X -0.173,Y -560.834,Z 1421.522,A 0.000,B 0.000,C 90.000,E1 129.930} C_DIS
LIN {X -0.042,Y -560.954,Z 1421.513,A 0.000,B 0.000,C 90.000,E1 128.257} C_DIS
LIN {X -0.002,Y -561.022,Z 1421.505,A 0.000,B 0.000,C 90.000,E1 126.870} C_DIS
LIN {X -0.303,Y -560.924,Z 1421.497,A 0.000,B 0.000,C 90.000,E1 125.518} C_DIS
LIN {X -0.245,Y -560.919,Z 1421.491,A 0.000,B 0.000,C 90.000,E1 124.405} C_DIS
LIN {X -0.098,Y -560.694,Z 1421.483,A 0.000,B 0.000,C 90.000,E1 123.007} C_DIS
LIN {X -0.056,Y -560.474,Z 1421.469,A 0.000,B 0.000,C 90.000,E1 120.512} C_DIS
LIN {X -0.043,Y -560.958,Z 1421.462,A 0.000,B 0.000,C 90.000,E1 119.127} C_DIS
LIN {X 0.208,Y -561.539,Z 1421.454,A 0.000,B 0.000,C 90.000,E1 117.719} C_DIS
LIN {X -0.020,Y -562.300,Z 1421.447,A 0.000,B 0.000,C 90.000,E1 116.360} C_DIS
LIN {X 0.096,Y -562.629,Z 1421.443,A 0.000,B 0.000,C 90.000,E1 115.796} C_DIS
LIN {X -0.117,Y -563.335,Z 1421.430,A 0.000,B 0.000,C 90.000,E1 113.334} C_DIS
LIN {X 0.107,Y -563.712,Z 1421.427,A 0.000,B 0.000,C 90.000,E1 112.898} C_DIS
LIN {X -0.188,Y -564.638,Z 1421.425,A 0.000,B 0.000,C 90.000,E1 112.514} C_DIS
LIN {X -0.096,Y -565.335,Z 1421.424,A 0.000,B 0.000,C 90.000,E1 112.333} C_DIS
LIN {X -0.194,Y -566.400,Z 1421.423,A 0.000,B 0.000,C 90.000,E1 112.206} C_DIS
LIN {X 0.079,Y -568.214,Z 1421.422,A 0.000,B 0.000,C 90.000,E1 111.972} C_DIS
LIN {X 0.042,Y -571.687,Z 1421.421,A 0.000,B 0.000,C 90.000,E1 111.770} C_DIS
LIN {X 0.299,Y -578.866,Z 1421.419,A 0.000,B 0.000,C 90.000,E1 111.408} C_DIS
LIN {X 0.004,Y -581.936,Z 1421.418,A 0.000,B 0.000,C 90.000,E1 111.280} C_DIS
LIN {X 0.144,Y -584.828,Z 1421.417,A 0.000,B 0.000,C 90.000,E1 111.099} C_DIS
LIN {X -0.141,Y -589.206,Z 1421.416,A 0.000,B 0.000,C 90.000,E1 110.844} C_DIS
LIN {X -0.328,Y -594.751,Z 1421.413,A 0.000,B 0.000,C 90.000,E1 110.429} C_DIS
LIN {X -0.063,Y -600.159,Z 1421.411,A 0.000,B 0.000,C 90.000,E1 109.939} C_DIS
LIN {X -0.283,Y -608.886,Z 1421.406,A 0.000,B 0.000,C 90.000,E1 109.087} C_DIS
LIN {X 0.036,Y -614.499,Z 1421.402,A 0.000,B 0.000,C 90.000,E1 108.417} C_DIS
LIN {X -0.242,Y -617.528,Z 1421.400,A 0.000,B 0.000,C 90.000,E1 108.055} C_DIS
LIN {X 0.063,Y -621.108,Z 1421.397,A 0.000,B 0.000,C 90.000,E1 107.511} C_DIS
LIN {X -0.183,Y -623.566,Z 1421.395,A 0.000,B 0.000,C 90.000,E1 107.149} C_DIS
LIN {X 0.179,Y -625.568,Z 1421.393,A 0.000,B 0.000,C 90.000,E1 106.732} C_DIS
LIN {X -0.241,Y -627.781,Z 1421.390,A 0.000,B 0.000,C 90.000,E1 106.260} C_DIS
LIN {X 0.159,Y -628.637,Z 1421.389,A 0.000,B 0.000,C 90.000,E1 105.969} C_DIS
LIN {X -0.263,Y -630.595,Z 1421.385,A 0.000,B 0.000,C 90.000,E1 105.245} C_DIS
LIN {X -0.036,Y -631.423,Z 1421.382,A 0.000,B 0.000,C 90.000,E1 104.717} C_DIS
LIN {X -0.205,Y -633.207,Z 1421.375,A 0.000,B 0.000,C 90.000,E1 103.467} C_DIS
LIN {X 0.043,Y -633.593,Z 1421.372,A 0.000,B 0.000,C 90.000,E1 102.939} C_DIS
LIN {X -0.022,Y -633.810,Z 1421.368,A 0.000,B 0.000,C 90.000,E1 102.187} C_DIS
LIN {X 0.237,Y -633.698,Z 1421.365,A 0.000,B 0.000,C 90.000,E1 101.658} C_DIS
LIN {X 0.307,Y -632.933,Z 1421.361,A 0.000,B 0.000,C 90.000,E1 100.894} C_DIS
LIN {X -0.068,Y -632.170,Z 1421.358,A 0.000,B 0.000,C 90.000,E1 100.423} C_DIS
LIN {X 0.060,Y -631.199,Z 1421.355,A 0.000,B 0.000,C 90.000,E1 99.905} C_DIS
LIN {X 0.291,Y -629.930,Z 1421.352,A 0.000,B 0.000,C 90.000,E1 99.378} C_DIS
LIN {X 0.204,Y -627.509,Z 1421.348,A 0.000,B 0.000,C 90.000,E1 98.624} C_DIS
LIN {X 0.310,Y -625.616,Z 1421.345,A 0.000,B 0.000,C 90.000,E1 98.106} C_DIS
LIN {X -0.211,Y -623.445,Z 1421.342,A 0.000,B 0.000,C 90.000,E1 97.644} C_DIS
LIN {X -0.204,Y -620.374,Z 1421.339,A 0.000,B 0.000,C 90.000,E1 97.004} C_DIS
LIN {X -0.145,Y -617.579,Z 1421.336,A 0.000,B 0.000,C 90.000,E1 96.486} C_DIS
LIN {X 0.180,Y -613.127,Z 1421.332,A 0.000,B 0.000,C 90.000,E1 95.682} C_DIS
LIN {X -0.146,Y -611.528,Z 1421.330,A 0.000,B 0.000,C 90.000,E1 95.454} C_DIS
LIN {X -0.262,Y -606.473,Z 1421.327,A 0.000,B 0.000,C 90.000,E1 94.816} C_DIS
LIN {X 0.255,Y -601.658,Z 1421.324,A 0.000,B 0.000,C 90.000,E1 94.245} C_DIS
LIN {X -0.028,Y -595.086,Z 1421.320,A 0.000,B 0.000,C 90.000,E1 93.669} C_DIS
LIN {X -0.125,Y -593.537,Z 1421.320,A 0.000,B 0.000,C 90.000,E1 93.555} C_DIS
LIN {X 0.049,Y -591.200,Z 1421.319,A 0.000,B 0.000,C 90.000,E1 93.326} C_DIS
LIN {X 0.052,Y -588.291,Z 1421.317,A 0.000,B 0.000,C 90.000,E1 93.094} C_DIS
LIN {X 0.168,Y -583.629,Z 1421.315,A 0.000,B 0.000,C 90.000,E1 92.751} C_DIS
LIN {X 0.011,Y -578.851,Z 1421.314,A 0.000,B 0.000,C 90.000,E1 92.465} C_DIS
LIN {X 0.184,Y -577.159,Z 1421.313,A 0.000,B 0.000,C 90.000,E1 92.350} C_DIS
LIN {X -0.062,Y -573.476,Z 1421.312,A 0.000,B 0.000,C 90.000,E1 92.064} C_DIS
LIN {X -0.100,Y -573.438,Z 1421.311,A 0.000,B 0.000,C 90.000,E1 92.064} C_DIS
LIN {X -0.017,Y -572.785,Z 1421.311,A 0.000,B 0.000,C 90.000,E1 91.892} C_DIS
LIN {X 0.142,Y -572.280,Z 1421.309,A 0.000,B 0.000,C 90.000,E1 91.604} C_DIS
LIN {X -0.155,Y -572.205,Z 1421.306,A 0.000,B 0.000,C 90.000,E1 91.088} C_DIS
LIN {X -0.178,Y -573.955,Z 1421.294,A 0.000,B 0.000,C 90.000,E1 88.912} C_DIS
LIN {X -0.157,Y -575.029,Z 1421.288,A 0.000,B 0.000,C 90.000,E1 87.822} C_DIS
LIN {X 0.034,Y -576.290,Z 1421.280,A 0.000,B 0.000,C 90.000,E1 86.445} C_DIS
LIN {X -0.146,Y -577.862,Z 1421.271,A 0.000,B 0.000,C 90.000,E1 84.837} C_DIS
LIN {X -0.027,Y -579.806,Z 1421.261,A 0.000,B 0.000,C 90.000,E1 82.932} C_DIS
LIN {X -0.228,Y -581.333,Z 1421.253,A 0.000,B 0.000,C 90.000,E1 81.602} C_DIS
LIN {X -0.181,Y -583.089,Z 1421.244,A 0.000,B 0.000,C 90.000,E1 79.982} C_DIS
LIN {X -0.134,Y -584.535,Z 1421.237,A 0.000,B 0.000,C 90.000,E1 78.634} C_DIS
LIN {X 0.272,Y -585.621,Z 1421.231,A 0.000,B 0.000,C 90.000,E1 77.521} C_DIS
LIN {X -0.201,Y -586.662,Z 1421.223,A 0.000,B 0.000,C 90.000,E1 76.228} C_DIS
LIN {X 0.050,Y -587.607,Z 1421.216,A 0.000,B 0.000,C 90.000,E1 74.866} C_DIS
LIN {X -0.251,Y -588.474,Z 1421.209,A 0.000,B 0.000,C 90.000,E1 73.559} C_DIS
LIN {X -0.130,Y -589.377,Z 1421.200,A 0.000,B 0.000,C 90.000,E1 71.945} C_DIS
LIN {X 0.058,Y -590.374,Z 1421.189,A 0.000,B 0.000,C 90.000,E1 70.061} C_DIS
LIN {X -0.286,Y -591.419,Z 1421.179,A 0.000,B 0.000,C 90.000,E1 68.230} C_DIS
LIN {X 0.275,Y -592.779,Z 1421.167,A 0.000,B 0.000,C 90.000,E1 66.049} C_DIS
LIN {X 0.050,Y -594.263,Z 1421.155,A 0.000,B 0.000,C 90.000,E1 63.948} C_DIS
LIN {X 0.131,Y -595.360,Z 1421.148,A 0.000,B 0.000,C 90.000,E1 62.615} C_DIS
LIN {X -0.116,Y -596.631,Z 1421.139,A 0.000,B 0.000,C 90.000,E1 61.051} C_DIS
LIN {X -0.127,Y -598.244,Z 1421.129,A 0.000,B 0.000,C 90.000,E1 59.203} C_DIS
LIN {X 0.293,Y -599.753,Z 1421.120,A 0.000,B 0.000,C 90.000,E1 57.582} C_DIS
LIN {X -0.005,Y -600.933,Z 1421.113,A 0.000,B 0.000,C 90.000,E1 56.294} C_DIS
LIN {X 0.298,Y -602.372,Z 1421.104,A 0.000,B 0.000,C 90.000,E1 54.689} C_DIS
LIN {X 0.141,Y -603.626,Z 1421.095,A 0.000,B 0.000,C 90.000,E1 53.130} C_DIS
LIN {X 0.110,Y -604.589,Z 1421.088,A 0.000,B 0.000,C 90.000,E1 51.823} C_DIS
LIN {X 0.092,Y -605.504,Z 1421.081,A 0.000,B 0.000,C 90.000,E1 50.517} C_DIS
LIN {X 0.007,Y -606.086,Z 1421.073,A 0.000,B 0.000,C 90.000,E1 49.218} C_DIS
LIN {X 0.134,Y -606.273,Z 1421.068,A 0.000,B 0.000,C 90.000,E1 48.162} C_DIS
LIN {X -0.133,Y -606.428,Z 1421.059,A 0.000,B 0.000,C 90.000,E1 46.620} C_DIS
LIN {X 0.150,Y -606.531,Z 1421.055,A 0.000,B 0.000,C 90.000,E1 45.810} C_DIS
LIN {X -0.132,Y -606.336,Z 1421.046,A 0.000,B 0.000,C 90.000,E1 44.271} C_DIS
LIN {X 0.013,Y -605.617,Z 1421.037,A 0.000,B 0.000,C 90.000,E1 42.690} C_DIS
LIN {X -0.069,Y -604.743,Z 1421.030,A 0.000,B 0.000,C 90.000,E1 41.391} C_DIS
LIN {X -0.217,Y -604.070,Z 1421.026,A 0.000,B 0.000,C 90.000,E1 40.620} C_DIS
LIN {X -0.122,Y -602.995,Z 1421.020,A 0.000,B 0.000,C 90.000,E1 39.564} C_DIS
LIN {X -0.051,Y -601.809,Z 1421.014,A 0.000,B 0.000,C 90.000,E1 38.508} C_DIS
LIN {X 0.347,Y -599.972,Z 1421.007,A 0.000,B 0.000,C 90.000,E1 37.156} C_DIS
LIN {X -0.004,Y -598.215,Z 1421.001,A 0.000,B 0.000,C 90.000,E1 36.137} C_DIS
LIN {X -0.132,Y -596.696,Z 1420.996,A 0.000,B 0.000,C 90.000,E1 35.358} C_DIS
LIN {X 0.100,Y -594.423,Z 1420.990,A 0.000,B 0.000,C 90.000,E1 34.278} C_DIS
LIN {X -0.068,Y -592.482,Z 1420.986,A 0.000,B 0.000,C 90.000,E1 33.499} C_DIS
LIN {X 0.117,Y -589.712,Z 1420.980,A 0.000,B 0.000,C 90.000,E1 32.418} C_DIS
LIN {X 0.195,Y -588.128,Z 1420.977,A 0.000,B 0.000,C 90.000,E1 31.878} C_DIS
LIN {X 0.317,Y -584.513,Z 1420.971,A 0.000,B 0.000,C 90.000,E1 30.797} C_DIS
LIN {X 0.062,Y -582.498,Z 1420.968,A 0.000,B 0.000,C 90.000,E1 30.285} C_DIS
LIN {X -0.046,Y -579.025,Z 1420.964,A 0.000,B 0.000,C 90.000,E1 29.489} C_DIS
LIN {X -0.119,Y -575.886,Z 1420.960,A 0.000,B 0.000,C 90.000,E1 28.821} C_DIS
LIN {X 0.196,Y -571.703,Z 1420.956,A 0.000,B 0.000,C 90.000,E1 27.975} C_DIS
LIN {X -0.131,Y -566.416,Z 1420.950,A 0.000,B 0.000,C 90.000,E1 27.052} C_DIS
LIN {X -0.085,Y -562.357,Z 1420.946,A 0.000,B 0.000,C 90.000,E1 26.360} C_DIS
LIN {X -0.171,Y -557.079,Z 1420.942,A 0.000,B 0.000,C 90.000,E1 25.540} C_DIS
LIN {X 0.310,Y -550.455,Z 1420.936,A 0.000,B 0.000,C 90.000,E1 24.515} C_DIS
LIN {X 0.216,Y -545.199,Z 1420.932,A 0.000,B 0.000,C 90.000,E1 23.823} C_DIS
LIN {X 0.207,Y -540.743,Z 1420.929,A 0.000,B 0.000,C 90.000,E1 23.259} C_DIS
LIN {X -0.041,Y -535.943,Z 1420.926,A 0.000,B 0.000,C 90.000,E1 22.717} C_DIS
LIN {X -0.065,Y -527.278,Z 1420.921,A 0.000,B 0.000,C 90.000,E1 21.716} C_DIS
LIN {X 0.167,Y -516.770,Z 1420.914,A 0.000,B 0.000,C 90.000,E1 20.556} C_DIS
LIN {X 0.196,Y -507.351,Z 1420.909,A 0.000,B 0.000,C 90.000,E1 19.577} C_DIS
LIN {X -0.092,Y -496.396,Z 1420.903,A 0.000,B 0.000,C 90.000,E1 18.489} C_DIS
LIN {X 0.168,Y -482.689,Z 1420.895,A 0.000,B 0.000,C 90.000,E1 17.040} C_DIS
LIN {X 0.018,Y -468.020,Z 1420.886,A 0.000,B 0.000,C 90.000,E1 15.481} C_DIS
LIN {X 0.138,Y -455.949,Z 1420.879,A 0.000,B 0.000,C 90.000,E1 14.120} C_DIS
LIN {X 0.144,Y -440.900,Z 1420.869,A 0.000,B 0.000,C 90.000,E1 12.411} C_DIS
LIN {X -0.160,Y -428.728,Z 1420.861,A 0.000,B 0.000,C 90.000,E1 11.007} C_DIS
LIN {X 0.039,Y -411.615,Z 1420.849,A 0.000,B 0.000,C 90.000,E1 8.803} C_DIS
LIN {X 0.085,Y -405.070,Z 1420.844,A 0.000,B 0.000,C 90.000,E1 7.936} C_DIS
LIN {X 0.166,Y -399.332,Z 1420.840,A 0.000,B 0.000,C 90.000,E1 7.239} C_DIS
LIN {X -0.048,Y -394.741,Z 1420.838,A 0.000,B 0.000,C 90.000,E1 6.777} C_DIS
LIN {X 0.086,Y -388.417,Z 1420.834,A 0.000,B 0.000,C 90.000,E1 6.144} C_DIS
LIN {X -0.022,Y -383.441,Z 1420.832,A 0.000,B 0.000,C 90.000,E1 5.739} C_DIS
LIN {X -0.164,Y -380.638,Z 1420.831,A 0.000,B 0.000,C 90.000,E1 5.568} C_DIS
LIN {X -0.198,Y -378.657,Z 1420.830,A 0.000,B 0.000,C 90.000,E1 5.511} C_DIS
LIN {X 0.152,Y -362.599,Z 1420.830,A 0.000,B 0.000,C 90.000,E1 5.454} C_DIS
LIN {X 0.014,Y -360.865,Z 1420.801,A 0.000,B 0.000,C 90.000,E1 0.115} C_DIS
LIN {X -0.053,Y -359.426,Z 1420.770,A 0.000,B 0.000,C 90.000,E1 354.546} C_DIS
LIN {X 0.070,Y -358.890,Z 1420.759,A 0.000,B 0.000,C 90.000,E1 352.648} C_DIS
LIN {X -0.020,Y -359.563,Z 1420.726,A 0.000,B 0.000,C 90.000,E1 346.645} C_DIS
LIN {X 0.001,Y -361.801,Z 1420.684,A 0.000,B 0.000,C 90.000,E1 339.135} C_DIS
LIN {X -0.154,Y -362.053,Z 1420.680,A 0.000,B 0.000,C 90.000,E1 338.411} C_DIS
LIN {X 0.189,Y -365.980,Z 1420.643,A 0.000,B 0.000,C 90.000,E1 331.641} C_DIS
LIN {X 0.029,Y -366.387,Z 1420.639,A 0.000,B 0.000,C 90.000,E1 330.923} C_DIS
LIN {X -0.031,Y -371.355,Z 1420.604,A 0.000,B 0.000,C 90.000,E1 324.642} C_DIS
LIN {X -0.043,Y -371.766,Z 1420.602,A 0.000,B 0.000,C 90.000,E1 324.276} C_DIS
LIN {X 0.013,Y -377.358,Z 1420.567,A 0.000,B 0.000,C 90.000,E1 318.038} C_DIS
LIN {X 0.012,Y -378.235,Z 1420.563,A 0.000,B 0.000,C 90.000,E1 317.310} C_DIS
LIN {X 0.002,Y -383.940,Z 1420.531,A 0.000,B 0.000,C 90.000,E1 311.515} C_DIS
LIN {X 0.088,Y -384.893,Z 1420.527,A 0.000,B 0.000,C 90.000,E1 310.782} C_DIS
LIN {X 0.262,Y -390.610,Z 1420.495,A 0.000,B 0.000,C 90.000,E1 305.025} C_DIS
LIN {X 0.106,Y -391.104,Z 1420.493,A 0.000,B 0.000,C 90.000,E1 304.692} C_DIS
LIN {X 0.022,Y -391.648,Z 1420.489,A 0.000,B 0.000,C 90.000,E1 303.992} C_DIS
LIN {X -0.080,Y -396.825,Z 1420.459,A 0.000,B 0.000,C 90.000,E1 298.693} C_DIS
LIN {X -0.210,Y -397.120,Z 1420.457,A 0.000,B 0.000,C 90.000,E1 298.359} C_DIS
LIN {X -0.055,Y -401.597,Z 1420.426,A 0.000,B 0.000,C 90.000,E1 292.717} C_DIS
LIN {X 0.222,Y -404.659,Z 1420.395,A 0.000,B 0.000,C 90.000,E1 287.094} C_DIS
LIN {X -0.079,Y -404.735,Z 1420.391,A 0.000,B 0.000,C 90.000,E1 286.441} C_DIS
LIN {X 0.214,Y -406.099,Z 1420.364,A 0.000,B 0.000,C 90.000,E1 281.535} C_DIS
LIN {X -0.176,Y -406.094,Z 1420.362,A 0.000,B 0.000,C 90.000,E1 281.243} C_DIS
LIN {X -0.097,Y -405.680,Z 1420.333,A 0.000,B 0.000,C 90.000,E1 276.024} C_DIS
LIN {X -0.165,Y -405.058,Z 1420.328,A 0.000,B 0.000,C 90.000,E1 274.992} C_DIS
LIN {X -0.060,Y -403.497,Z 1420.304,A 0.000,B 0.000,C 90.000,E1 270.802} C_DIS
LIN {X -0.092,Y -403.288,Z 1420.302,A 0.000,B 0.000,C 90.000,E1 270.458} C_DIS
LIN {X 0.091,Y -398.931,Z 1420.271,A 0.000,B 0.000,C 90.000,E1 264.837} C_DIS
LIN {X -0.040,Y -393.108,Z 1420.242,A 0.000,B 0.000,C 90.000,E1 259.567} C_DIS
LIN {X -0.079,Y -392.835,Z 1420.240,A 0.000,B 0.000,C 90.000,E1 259.218} C_DIS
LIN {X 0.034,Y -385.993,Z 1420.212,A 0.000,B 0.000,C 90.000,E1 254.212} C_DIS
LIN {X -0.026,Y -385.267,Z 1420.208,A 0.000,B 0.000,C 90.000,E1 253.504} C_DIS
LIN {X -0.004,Y -384.768,Z 1420.206,A 0.000,B 0.000,C 90.000,E1 253.142} C_DIS
LIN {X 0.221,Y -377.973,Z 1420.182,A 0.000,B 0.000,C 90.000,E1 248.773} C_DIS
LIN {X -0.044,Y -376.233,Z 1420.174,A 0.000,B 0.000,C 90.000,E1 247.358} C_DIS
LIN {X 0.057,Y -374.944,Z 1420.170,A 0.000,B 0.000,C 90.000,E1 246.613} C_DIS
LIN {X -0.208,Y -368.417,Z 1420.148,A 0.000,B 0.000,C 90.000,E1 242.615} C_DIS
LIN {X 0.097,Y -366.047,Z 1420.137,A 0.000,B 0.000,C 90.000,E1 240.717} C_DIS
LIN {X 0.004,Y -359.196,Z 1420.115,A 0.000,B 0.000,C 90.000,E1 236.628} C_DIS
LIN {X 0.021,Y -355.842,Z 1420.100,A 0.000,B 0.000,C 90.000,E1 233.989} C_DIS
LIN {X -0.173,Y -348.793,Z 1420.075,A 0.000,B 0.000,C 90.000,E1 229.461} C_DIS
LIN {X -0.097,Y -346.185,Z 1420.062,A 0.000,B 0.000,C 90.000,E1 227.148} C_DIS
LIN {X -0.088,Y -345.065,Z 1420.058,A 0.000,B 0.000,C 90.000,E1 226.377} C_DIS
LIN {X 0.094,Y -338.586,Z 1420.030,A 0.000,B 0.000,C 90.000,E1 221.310} C_DIS
LIN {X 0.094,Y -336.840,Z 1420.019,A 0.000,B 0.000,C 90.000,E1 219.358} C_DIS
LIN {X 0.014,Y -330.861,Z 1419.988,A 0.000,B 0.000,C 90.000,E1 213.865} C_DIS
LIN {X 0.149,Y -329.296,Z 1419.975,A 0.000,B 0.000,C 90.000,E1 211.465} C_DIS
LIN {X -0.154,Y -324.669,Z 1419.942,A 0.000,B 0.000,C 90.000,E1 205.540} C_DIS
LIN {X 0.174,Y -323.837,Z 1419.928,A 0.000,B 0.000,C 90.000,E1 203.078} C_DIS
LIN {X -0.017,Y -321.124,Z 1419.881,A 0.000,B 0.000,C 90.000,E1 194.662} C_DIS
LIN {X 0.138,Y -320.932,Z 1419.877,A 0.000,B 0.000,C 90.000,E1 193.828} C_DIS
LIN {X -0.076,Y -321.562,Z 1419.832,A 0.000,B 0.000,C 90.000,E1 185.796} C_DIS
LIN {X -0.143,Y -324.415,Z 1419.790,A 0.000,B 0.000,C 90.000,E1 178.165} C_DIS
LIN {X -0.141,Y -325.376,Z 1419.783,A 0.000,B 0.000,C 90.000,E1 176.963} C_DIS
LIN {X 0.000,Y -326.421,Z 1419.770,A 0.000,B 0.000,C 90.000,E1 174.546} C_DIS
LIN {X -0.019,Y -344.144,Z 1419.770,A 0.000,B 0.000,C 90.000,E1 174.546} C_DIS
LIN {X -0.104,Y -345.508,Z 1419.769,A 0.000,B 0.000,C 90.000,E1 174.489} C_DIS
LIN {X 0.056,Y -346.257,Z 1419.768,A 0.000,B 0.000,C 90.000,E1 174.261} C_DIS
LIN {X 0.174,Y -346.051,Z 1419.766,A 0.000,B 0.000,C 90.000,E1 173.856} C_DIS
LIN {X 0.035,Y -344.292,Z 1419.762,A 0.000,B 0.000,C 90.000,E1 173.109} C_DIS
LIN {X -0.073,Y -342.002,Z 1419.758,A 0.000,B 0.000,C 90.000,E1 172.356} C_DIS
LIN {X 0.041,Y -341.165,Z 1419.754,A 0.000,B 0.000,C 90.000,E1 171.659} C_DIS
LIN {X -0.143,Y -341.085,Z 1419.753,A 0.000,B 0.000,C 90.000,E1 171.602} C_DIS
LIN {X 0.176,Y -341.084,Z 1419.753,A 0.000,B 0.000,C 90.000,E1 171.546} C_DIS
LIN {X 0.007,Y -341.997,Z 1419.751,A 0.000,B 0.000,C 90.000,E1 171.141} C_DIS
LIN {X -0.160,Y -342.108,Z 1419.750,A 0.000,B 0.000,C 90.000,E1 171.084} C_DIS
LIN {X 0.152,Y -342.114,Z 1419.750,A 0.000,B 0.000,C 90.000,E1 171.027} C_DIS
LIN {X -0.098,Y -345.214,Z 1419.747,A 0.000,B 0.000,C 90.000,E1 170.443} C_DIS
LIN {X 0.106,Y -349.167,Z 1419.743,A 0.000,B 0.000,C 90.000,E1 169.746} C_DIS
LIN {X 0.154,Y -360.025,Z 1419.735,A 0.000,B 0.000,C 90.000,E1 168.229} C_DIS
LIN {X -0.089,Y -374.408,Z 1419.725,A 0.000,B 0.000,C 90.000,E1 166.464} C_DIS
LIN {X -0.130,Y -386.006,Z 1419.718,A 0.000,B 0.000,C 90.000,E1 165.172} C_DIS
LIN {X 0.106,Y -395.162,Z 1419.712,A 0.000,B 0.000,C 90.000,E1 164.212} C_DIS
LIN {X -0.098,Y -409.074,Z 1419.705,A 0.000,B 0.000,C 90.000,E1 162.960} C_DIS
LIN {X -0.086,Y -426.151,Z 1419.697,A 0.000,B 0.000,C 90.000,E1 161.511} C_DIS
LIN {X -0.024,Y -439.895,Z 1419.691,A 0.000,B 0.000,C 90.000,E1 160.369} C_DIS
LIN {X 0.213,Y -447.582,Z 1419.687,A 0.000,B 0.000,C 90.000,E1 159.699} C_DIS
LIN {X -0.209,Y -459.841,Z 1419.682,A 0.000,B 0.000,C 90.000,E1 158.720} C_DIS
LIN {X 0.011,Y -470.466,Z 1419.677,A 0.000,B 0.000,C 90.000,E1 157.794} C_DIS
LIN {X 0.087,Y -480.876,Z 1419.672,A 0.000,B 0.000,C 90.000,E1 156.869} C_DIS
LIN {X -0.085,Y -488.111,Z 1419.668,A 0.000,B 0.000,C 90.000,E1 156.230} C_DIS
LIN {X 0.046,Y -495.216,Z 1419.664,A 0.000,B 0.000,C 90.000,E1 155.537} C_DIS
LIN {X 0.192,Y -500.716,Z 1419.661,A 0.000,B 0.000,C 90.000,E1 154.973} C_DIS
LIN {X 0.100,Y -507.428,Z 1419.657,A 0.000,B 0.000,C 90.000,E1 154.280} C_DIS
LIN {X 0.058,Y -513.746,Z 1419.653,A 0.000,B 0.000,C 90.000,E1 153.563} C_DIS
LIN {X 0.010,Y -517.407,Z 1419.651,A 0.000,B 0.000,C 90.000,E1 153.127} C_DIS
LIN {X -0.065,Y -522.790,Z 1419.647,A 0.000,B 0.000,C 90.000,E1 152.410} C_DIS
LIN {X -0.085,Y -525.796,Z 1419.644,A 0.000,B 0.000,C 90.000,E1 151.975} C_DIS
LIN {X 0.004,Y -529.372,Z 1419.641,A 0.000,B 0.000,C 90.000,E1 151.385} C_DIS
LIN {X 0.123,Y -532.604,Z 1419.638,A 0.000,B 0.000,C 90.000,E1 150.795} C_DIS
LIN {X 0.121,Y -536.041,Z 1419.634,A 0.000,B 0.000,C 90.000,E1 150.078} C_DIS
LIN {X -0.317,Y -539.015,Z 1419.630,A 0.000,B 0.000,C 90.000,E1 149.410} C_DIS
LIN {X 0.146,Y -541.192,Z 1419.627,A 0.000,B 0.000,C 90.000,E1 148.791} C_DIS
LIN {X -0.116,Y -543.091,Z 1419.624,A 0.000,B 0.000,C 90.000,E1 148.250} C_DIS
LIN {X 0.123,Y -545.625,Z 1419.619,A 0.000,B 0.000,C 90.000,E1 147.375} C_DIS
LIN {X -0.109,Y -547.144,Z 1419.616,A 0.000,B 0.000,C 90.000,E1 146.834} C_DIS
LIN {X 0.213,Y -549.757,Z 1419.609,A 0.000,B 0.000,C 90.000,E1 145.674} C_DIS
LIN {X 0.058,Y -551.469,Z 1419.605,A 0.000,B 0.000,C 90.000,E1 144.848} C_DIS
LIN {X 0.239,Y -552.865,Z 1419.600,A 0.000,B 0.000,C 90.000,E1 143.989} C_DIS
LIN {X -0.268,Y -554.261,Z 1419.594,A 0.000,B 0.000,C 90.000,E1 142.924} C_DIS
LIN {X -0.055,Y -555.157,Z 1419.589,A 0.000,B 0.000,C 90.000,E1 142.065} C_DIS
LIN {X 0.308,Y -556.701,Z 1419.580,A 0.000,B 0.000,C 90.000,E1 140.356} C_DIS
LIN {X -0.235,Y -557.614,Z 1419.574,A 0.000,B 0.000,C 90.000,E1 139.299} C_DIS
LIN {X 0.095,Y -558.534,Z 1419.566,A 0.000,B 0.000,C 90.000,E1 137.877} C_DIS
LIN {X -0.272,Y -559.595,Z 1419.555,A 0.000,B 0.000,C 90.000,E1 135.972} C_DIS
LIN {X 0.046,Y -560.132,Z 1419.548,A 0.000,B 0.000,C 90.000,E1 134.555} C_DIS
LIN {X 0.040,Y -560.528,Z 1419.538,A 0.000,B 0.000,C 90.000,E1 132.894} C_DIS
LIN {X -0.004,Y -560.659,Z 1419.531,A 0.000,B 0.000,C 90.000,E1 131.515} C_DIS
LIN {X 0.043,Y -560.765,Z 1419.521,A 0.000,B 0.000,C 90.000,E1 129.850} C_DIS
LIN {X 0.171,Y -560.932,Z 1419.512,A 0.000,B 0.000,C 90.000,E1 128.177} C_DIS
LIN {X 0.208,Y -560.991,Z 1419.505,A 0.000,B 0.000,C 90.000,E1 126.790} C_DIS
LIN {X -0.002,Y -560.901,Z 1419.495,A 0.000,B 0.000,C 90.000,E1 125.152} C_DIS
LIN {X 0.052,Y -560.891,Z 1419.489,A 0.000,B 0.000,C 90.000,E1 124.040} C_DIS
LIN {X -0.203,Y -560.697,Z 1419.483,A 0.000,B 0.000,C 90.000,E1 122.959} C_DIS
LIN {X 0.060,Y -560.499,Z 1419.471,A 0.000,B 0.000,C 90.000,E1 120.718} C_DIS
LIN {X 0.076,Y -561.088,Z 1419.463,A 0.000,B 0.000,C 90.000,E1 119.333} C_DIS
LIN {X -0.101,Y -561.937,Z 1419.454,A 0.000,B 0.000,C 90.000,E1 117.692} C_DIS
LIN {X 0.003,Y -562.566,Z 1419.451,A 0.000,B 0.000,C 90.000,E1 117.129} C_DIS
LIN {X -0.147,Y -563.066,Z 1419.450,A 0.000,B 0.000,C 90.000,E1 117.001} C_DIS
LIN {X -0.072,Y -563.776,Z 1419.447,A 0.000,B 0.000,C 90.000,E1 116.437} C_DIS
LIN {X 0.136,Y -563.807,Z 1419.447,A 0.000,B 0.000,C 90.000,E1 116.411} C_DIS
LIN {X 0.125,Y -564.748,Z 1419.446,A 0.000,B 0.000,C 90.000,E1 116.283} C_DIS
LIN {X 0.028,Y -565.576,Z 1419.445,A 0.000,B 0.000,C 90.000,E1 116.155} C_DIS
LIN {X -0.162,Y -568.614,Z 1419.444,A 0.000,B 0.000,C 90.000,E1 115.899} C_DIS
LIN {X 0.337,Y -570.186,Z 1419.442,A 0.000,B 0.000,C 90.000,E1 115.591} C_DIS
LIN {X -0.011,Y -571.781,Z 1419.439,A 0.000,B 0.000,C 90.000,E1 115.079} C_DIS
LIN {X -0.096,Y -571.800,Z 1419.439,A 0.000,B 0.000,C 90.000,E1 114.951} C_DIS
LIN {X -0.259,Y -570.688,Z 1419.438,A 0.000,B 0.000,C 90.000,E1 114.899} C_DIS
LIN {X -0.081,Y -568.625,Z 1419.438,A 0.000,B 0.000,C 90.000,E1 114.847} C_DIS
LIN {X 0.159,Y -567.204,Z 1419.436,A 0.000,B 0.000,C 90.000,E1 114.515} C_DIS
LIN {X -0.310,Y -564.437,Z 1419.434,A 0.000,B 0.000,C 90.000,E1 114.207} C_DIS
LIN {X 0.164,Y -564.415,Z 1419.434,A 0.000,B 0.000,C 90.000,E1 114.155} C_DIS
LIN {X 0.310,Y -564.595,Z 1419.433,A 0.000,B 0.000,C 90.000,E1 113.951} C_DIS
LIN {X 0.022,Y -563.940,Z 1419.431,A 0.000,B 0.000,C 90.000,E1 113.567} C_DIS
LIN {X -0.070,Y -564.428,Z 1419.428,A 0.000,B 0.000,C 90.000,E1 113.025} C_DIS
LIN {X -0.167,Y -564.782,Z 1419.427,A 0.000,B 0.000,C 90.000,E1 112.898} C_DIS
LIN {X 0.238,Y -566.010,Z 1419.425,A 0.000,B 0.000,C 90.000,E1 112.514} C_DIS
LIN {X 0.098,Y -566.446,Z 1419.425,A 0.000,B 0.000,C 90.000,E1 112.461} C_DIS
LIN {X -0.052,Y -568.870,Z 1419.423,A 0.000,B 0.000,C 90.000,E1 112.206} C_DIS
LIN {X -0.065,Y -572.555,Z 1419.422,A 0.000,B 0.000,C 90.000,E1 111.972} C_DIS
LIN {X 0.024,Y -580.437,Z 1419.420,A 0.000,B 0.000,C 90.000,E1 111.589} C_DIS
LIN {X 0.220,Y -583.642,Z 1419.419,A 0.000,B 0.000,C 90.000,E1 111.408} C_DIS
LIN {X -0.200,Y -589.539,Z 1419.417,A 0.000,B 0.000,C 90.000,E1 111.099} C_DIS
LIN {X -0.045,Y -593.501,Z 1419.416,A 0.000,B 0.000,C 90.000,E1 110.791} C_DIS
LIN {X 0.287,Y -597.505,Z 1419.414,A 0.000,B 0.000,C 90.000,E1 110.429} C_DIS
LIN {X -0.190,Y -601.493,Z 1419.412,A 0.000,B 0.000,C 90.000,E1 110.120} C_DIS
LIN {X -0.179,Y -606.580,Z 1419.409,A 0.000,B 0.000,C 90.000,E1 109.631} C_DIS
LIN {X 0.199,Y -611.448,Z 1419.406,A 0.000,B 0.000,C 90.000,E1 109.087} C_DIS
LIN {X -0.081,Y -615.948,Z 1419.403,A 0.000,B 0.000,C 90.000,E1 108.598} C_DIS
LIN {X 0.214,Y -620.126,Z 1419.401,A 0.000,B 0.000,C 90.000,E1 108.055} C_DIS
LIN {X 0.321,Y -625.173,Z 1419.396,A 0.000,B 0.000,C 90.000,E1 107.275} C_DIS
LIN {X -0.112,Y -628.488,Z 1419.393,A 0.000,B 0.000,C 90.000,E1 106.677} C_DIS
LIN {X -0.314,Y -629.535,Z 1419.391,A 0.000,B 0.000,C 90.000,E1 106.441} C_DIS
LIN {X 0.073,Y -631.208,Z 1419.388,A 0.000,B 0.000,C 90.000,E1 105.898} C_DIS
LIN {X -0.310,Y -632.512,Z 1419.386,A 0.000,B 0.000,C 90.000,E1 105.426} C_DIS
LIN {X -0.070,Y -633.373,Z 1419.383,A 0.000,B 0.000,C 90.000,E1 104.898} C_DIS
LIN {X -0.022,Y -634.868,Z 1419.377,A 0.000,B 0.000,C 90.000,E1 103.883} C_DIS
LIN {X 0.062,Y -635.593,Z 1419.373,A 0.000,B 0.000,C 90.000,E1 103.119} C_DIS
LIN {X 0.330,Y -635.880,Z 1419.370,A 0.000,B 0.000,C 90.000,E1 102.591} C_DIS
LIN {X -0.022,Y -636.039,Z 1419.367,A 0.000,B 0.000,C 90.000,E1 102.119} C_DIS
LIN {X 0.248,Y -635.867,Z 1419.365,A 0.000,B 0.000,C 90.000,E1 101.591} C_DIS
LIN {X -0.231,Y -635.332,Z 1419.362,A 0.000,B 0.000,C 90.000,E1 101.130} C_DIS
LIN {X -0.147,Y -634.155,Z 1419.358,A 0.000,B 0.000,C 90.000,E1 100.366} C_DIS
LIN {X -0.004,Y -633.150,Z 1419.355,A 0.000,B 0.000,C 90.000,E1 99.849} C_DIS
LIN {X 0.241,Y -631.901,Z 1419.352,A 0.000,B 0.000,C 90.000,E1 99.321} C_DIS
LIN {X -0.247,Y -630.368,Z 1419.349,A 0.000,B 0.000,C 90.000,E1 98.859} C_DIS
LIN {X -0.119,Y -628.594,Z 1419.346,A 0.000,B 0.000,C 90.000,E1 98.341} C_DIS
LIN {X 0.087,Y -626.513,Z 1419.344,A 0.000,B 0.000,C 90.000,E1 97.814} C_DIS
LIN {X 0.189,Y -624.147,Z 1419.341,A 0.000,B 0.000,C 90.000,E1 97.296} C_DIS
LIN {X 0.121,Y -620.966,Z 1419.337,A 0.000,B 0.000,C 90.000,E1 96.663} C_DIS
LIN {X -0.273,Y -618.831,Z 1419.335,A 0.000,B 0.000,C 90.000,E1 96.315} C_DIS
LIN {X 0.070,Y -614.329,Z 1419.331,A 0.000,B 0.000,C 90.000,E1 95.511} C_DIS
LIN {X -0.194,Y -612.589,Z 1419.329,A 0.000,B 0.000,C 90.000,E1 95.277} C_DIS
LIN {X -0.077,Y -609.644,Z 1419.327,A 0.000,B 0.000,C 90.000,E1 94.878} C_DIS
LIN {X -0.260,Y -603.914,Z 1419.323,A 0.000,B 0.000,C 90.000,E1 94.245} C_DIS
LIN {X 0.186,Y -598.725,Z 1419.321,A 0.000,B 0.000,C 90.000,E1 93.726} C_DIS
LIN {X 0.185,Y -597.531,Z 1419.320,A 0.000,B 0.000,C 90.000,E1 93.612} C_DIS
LIN {X 0.240,Y -593.420,Z 1419.318,A 0.000,B 0.000,C 90.000,E1 93.269} C_DIS
LIN {X 0.199,Y -590.876,Z 1419.317,A 0.000,B 0.000,C 90.000,E1 93.037} C_DIS
LIN {X -0.110,Y -583.265,Z 1419.314,A 0.000,B 0.000,C 90.000,E1 92.522} C_DIS
LIN {X -0.098,Y -578.266,Z 1419.312,A 0.000,B 0.000,C 90.000,E1 92.236} C_DIS
LIN {X 0.147,Y -576.915,Z 1419.312,A 0.000,B 0.000,C 90.000,E1 92.121} C_DIS
LIN {X 0.174,Y -573.539,Z 1419.310,A 0.000,B 0.000,C 90.000,E1 91.835} C_DIS
LIN {X 0.136,Y -573.496,Z 1419.310,A 0.000,B 0.000,C 90.000,E1 91.835} C_DIS
LIN {X 0.103,Y -572.796,Z 1419.309,A 0.000,B 0.000,C 90.000,E1 91.661} C_DIS
LIN {X 0.181,Y -572.385,Z 1419.308,A 0.000,B 0.000,C 90.000,E1 91.375} C_DIS
LIN {X -0.115,Y -572.365,Z 1419.305,A 0.000,B 0.000,C 90.000,E1 90.859} C_DIS
LIN {X -0.276,Y -573.914,Z 1419.294,A 0.000,B 0.000,C 90.000,E1 88.969} C_DIS
LIN {X -0.109,Y -575.229,Z 1419.287,A 0.000,B 0.000,C 90.000,E1 87.593} C_DIS
LIN {X 0.227,Y -576.735,Z 1419.278,A 0.000,B 0.000,C 90.000,E1 85.931} C_DIS
LIN {X 0.103,Y -578.355,Z 1419.269,A 0.000,B 0.000,C 90.000,E1 84.318} C_DIS
LIN {X -0.197,Y -580.687,Z 1419.256,A 0.000,B 0.000,C 90.000,E1 82.186} C_DIS
LIN {X 0.041,Y -581.874,Z 1419.250,A 0.000,B 0.000,C 90.000,E1 81.084} C_DIS
LIN {X -0.041,Y -583.351,Z 1419.243,A 0.000,B 0.000,C 90.000,E1 79.746} C_DIS
LIN {X 0.139,Y -585.094,Z 1419.234,A 0.000,B 0.000,C 90.000,E1 78.117} C_DIS
LIN {X -0.029,Y -586.029,Z 1419.228,A 0.000,B 0.000,C 90.000,E1 77.061} C_DIS
LIN {X 0.205,Y -587.069,Z 1419.221,A 0.000,B 0.000,C 90.000,E1 75.700} C_DIS
LIN {X 0.139,Y -588.149,Z 1419.212,A 0.000,B 0.000,C 90.000,E1 74.102} C_DIS
LIN {X 0.008,Y -588.918,Z 1419.204,A 0.000,B 0.000,C 90.000,E1 72.779} C_DIS
LIN {X -0.209,Y -589.400,Z 1419.200,A 0.000,B 0.000,C 90.000,E1 72.000} C_DIS
LIN {X 0.216,Y -590.536,Z 1419.188,A 0.000,B 0.000,C 90.000,E1 69.826} C_DIS
LIN {X 0.087,Y -591.563,Z 1419.178,A 0.000,B 0.000,C 90.000,E1 67.975} C_DIS
LIN {X 0.219,Y -592.786,Z 1419.167,A 0.000,B 0.000,C 90.000,E1 66.102} C_DIS
LIN {X -0.258,Y -594.304,Z 1419.156,A 0.000,B 0.000,C 90.000,E1 64.024} C_DIS
LIN {X 0.089,Y -595.391,Z 1419.148,A 0.000,B 0.000,C 90.000,E1 62.666} C_DIS
LIN {X -0.149,Y -596.665,Z 1419.139,A 0.000,B 0.000,C 90.000,E1 61.101} C_DIS
LIN {X -0.149,Y -598.282,Z 1419.129,A 0.000,B 0.000,C 90.000,E1 59.253} C_DIS
LIN {X 0.192,Y -600.019,Z 1419.119,A 0.000,B 0.000,C 90.000,E1 57.375} C_DIS
LIN {X -0.101,Y -601.193,Z 1419.112,A 0.000,B 0.000,C 90.000,E1 56.087} C_DIS
LIN {X -0.044,Y -602.417,Z 1419.104,A 0.000,B 0.000,C 90.000,E1 54.769} C_DIS
LIN {X -0.206,Y -603.670,Z 1419.096,A 0.000,B 0.000,C 90.000,E1 53.210} C_DIS
LIN {X -0.239,Y -604.636,Z 1419.088,A 0.000,B 0.000,C 90.000,E1 51.904} C_DIS
LIN {X 0.126,Y -605.563,Z 1419.081,A 0.000,B 0.000,C 90.000,E1 50.561} C_DIS
LIN {X -0.144,Y -606.064,Z 1419.075,A 0.000,B 0.000,C 90.000,E1 49.542} C_DIS
LIN {X -0.022,Y -606.339,Z 1419.069,A 0.000,B 0.000,C 90.000,E1 48.485} C_DIS
LIN {X -0.068,Y -606.556,Z 1419.059,A 0.000,B 0.000,C 90.000,E1 46.662} C_DIS
LIN {X 0.044,Y -606.589,Z 1419.053,A 0.000,B 0.000,C 90.000,E1 45.607} C_DIS
LIN {X 0.377,Y -606.434,Z 1419.046,A 0.000,B 0.000,C 90.000,E1 44.271} C_DIS
LIN {X -0.139,Y -605.842,Z 1419.039,A 0.000,B 0.000,C 90.000,E1 43.014} C_DIS
LIN {X -0.063,Y -605.237,Z 1419.033,A 0.000,B 0.000,C 90.000,E1 41.962} C_DIS
LIN {X 0.042,Y -604.480,Z 1419.027,A 0.000,B 0.000,C 90.000,E1 40.906} C_DIS
LIN {X 0.139,Y -603.426,Z 1419.021,A 0.000,B 0.000,C 90.000,E1 39.850} C_DIS
LIN {X 0.090,Y -602.026,Z 1419.014,A 0.000,B 0.000,C 90.000,E1 38.543} C_DIS
LIN {X 0.024,Y -600.207,Z 1419.007,A 0.000,B 0.000,C 90.000,E1 37.237} C_DIS
LIN {X 0.164,Y -598.486,Z 1419.001,A 0.000,B 0.000,C 90.000,E1 36.171} C_DIS
LIN {X 0.044,Y -596.997,Z 1418.997,A 0.000,B 0.000,C 90.000,E1 35.391} C_DIS
LIN {X 0.132,Y -594.761,Z 1418.991,A 0.000,B 0.000,C 90.000,E1 34.326} C_DIS
LIN {X -0.364,Y -592.830,Z 1418.986,A 0.000,B 0.000,C 90.000,E1 33.579} C_DIS
LIN {X 0.147,Y -590.119,Z 1418.980,A 0.000,B 0.000,C 90.000,E1 32.467} C_DIS
LIN {X 0.225,Y -588.546,Z 1418.978,A 0.000,B 0.000,C 90.000,E1 31.926} C_DIS
LIN {X 0.047,Y -584.945,Z 1418.972,A 0.000,B 0.000,C 90.000,E1 30.875} C_DIS
LIN {X 0.091,Y -582.978,Z 1418.969,A 0.000,B 0.000,C 90.000,E1 30.335} C_DIS
LIN {X -0.038,Y -581.940,Z 1418.967,A 0.000,B 0.000,C 90.000,E1 30.079} C_DIS
LIN {X -0.015,Y -577.109,Z 1418.961,A 0.000,B 0.000,C 90.000,E1 28.999} C_DIS
LIN {X 0.040,Y -573.013,Z 1418.957,A 0.000,B 0.000,C 90.000,E1 28.180} C_DIS
LIN {X -0.097,Y -569.347,Z 1418.953,A 0.000,B 0.000,C 90.000,E1 27.513} C_DIS
LIN {X 0.139,Y -564.705,Z 1418.948,A 0.000,B 0.000,C 90.000,E1 26.668} C_DIS
LIN {X 0.171,Y -560.477,Z 1418.944,A 0.000,B 0.000,C 90.000,E1 25.976} C_DIS
LIN {X 0.063,Y -555.049,Z 1418.940,A 0.000,B 0.000,C 90.000,E1 25.155} C_DIS
LIN {X 0.014,Y -550.249,Z 1418.936,A 0.000,B 0.000,C 90.000,E1 24.463} C_DIS
LIN {X -0.075,Y -544.936,Z 1418.932,A 0.000,B 0.000,C 90.000,E1 23.770} C_DIS
LIN {X -0.213,Y -539.271,Z 1418.928,A 0.000,B 0.000,C 90.000,E1 23.078} C_DIS
LIN {X 0.247,Y -528.497,Z 1418.921,A 0.000,B 0.000,C 90.000,E1 21.770} C_DIS
LIN {X -0.136,Y -521.954,Z 1418.917,A 0.000,B 0.000,C 90.000,E1 21.099} C_DIS
LIN {X -0.076,Y -514.011,Z 1418.912,A 0.000,B 0.000,C 90.000,E1 20.248} C_DIS
LIN {X 0.031,Y -504.588,Z 1418.907,A 0.000,B 0.000,C 90.000,E1 19.268} C_DIS
LIN {X -0.047,Y -496.902,Z 1418.903,A 0.000,B 0.000,C 90.000,E1 18.489} C_DIS
LIN {X -0.016,Y -484.611,Z 1418.896,A 0.000,B 0.000,C 90.000,E1 17.221} C_DIS
LIN {X 0.091,Y -475.191,Z 1418.890,A 0.000,B 0.000,C 90.000,E1 16.205} C_DIS
LIN {X -0.208,Y -459.136,Z 1418.880,A 0.000,B 0.000,C 90.000,E1 14.481} C_DIS
LIN {X -0.075,Y -448.225,Z 1418.874,A 0.000,B 0.000,C 90.000,E1 13.244} C_DIS
LIN {X -0.027,Y -435.988,Z 1418.866,A 0.000,B 0.000,C 90.000,E1 11.827} C_DIS
LIN {X 0.207,Y -415.887,Z 1418.852,A 0.000,B 0.000,C 90.000,E1 9.321} C_DIS
LIN {X 0.115,Y -403.250,Z 1418.843,A 0.000,B 0.000,C 90.000,E1 7.644} C_DIS
LIN {X 0.108,Y -397.801,Z 1418.839,A 0.000,B 0.000,C 90.000,E1 6.947} C_DIS
LIN {X -0.173,Y -390.522,Z 1418.834,A 0.000,B 0.000,C 90.000,E1 6.144} C_DIS
LIN {X -0.006,Y -386.074,Z 1418.831,A 0.000,B 0.000,C 90.000,E1 5.625} C_DIS
LIN {X -0.108,Y -381.190,Z 1418.828,A 0.000,B 0.000,C 90.000,E1 5.049} C_DIS
LIN {X -0.022,Y -379.474,Z 1418.826,A 0.000,B 0.000,C 90.000,E1 4.759} C_DIS
LIN {X -0.114,Y -378.358,Z 1418.826,A 0.000,B 0.000,C 90.000,E1 4.645} C_DIS
LIN {X -0.071,Y -377.716,Z 1418.825,A 0.000,B 0.000,C 90.000,E1 4.588} C_DIS
LIN {X 0.016,Y -376.646,Z 1418.825,A 0.000,B 0.000,C 90.000,E1 4.531} C_DIS
LIN {X -0.007,Y -362.061,Z 1418.825,A 0.000,B 0.000,C 90.000,E1 4.531} C_DIS
LIN {X 0.085,Y -360.907,Z 1418.802,A 0.000,B 0.000,C 90.000,E1 0.344} C_DIS
LIN {X -0.058,Y -360.492,Z 1418.797,A 0.000,B 0.000,C 90.000,E1 359.427} C_DIS
LIN {X -0.053,Y -359.426,Z 1418.770,A 0.000,B 0.000,C 90.000,E1 354.546} C_DIS
LIN {X 0.070,Y -358.890,Z 1418.759,A 0.000,B 0.000,C 90.000,E1 352.648} C_DIS
LIN {X -0.020,Y -359.563,Z 1418.726,A 0.000,B 0.000,C 90.000,E1 346.645} C_DIS
LIN {X 0.001,Y -361.801,Z 1418.684,A 0.000,B 0.000,C 90.000,E1 339.135} C_DIS
LIN {X -0.154,Y -362.053,Z 1418.680,A 0.000,B 0.000,C 90.000,E1 338.411} C_DIS
LIN {X 0.189,Y -365.980,Z 1418.643,A 0.000,B 0.000,C 90.000,E1 331.641} C_DIS
LIN {X 0.029,Y -366.387,Z 1418.639,A 0.000,B 0.000,C 90.000,E1 330.923} C_DIS
LIN {X -0.031,Y -371.355,Z 1418.604,A 0.000,B 0.000,C 90.000,E1 324.642} C_DIS
LIN {X -0.043,Y -371.766,Z 1418.602,A 0.000,B 0.000,C 90.000,E1 324.276} C_DIS
LIN {X 0.013,Y -377.358,Z 1418.567,A 0.000,B 0.000,C 90.000,E1 318.038} C_DIS
LIN {X 0.012,Y -378.235,Z 1418.563,A 0.000,B 0.000,C 90.000,E1 317.310} C_DIS
LIN {X 0.002,Y -383.940,Z 1418.531,A 0.000,B 0.000,C 90.000,E1 311.515} C_DIS
LIN {X 0.088,Y -384.893,Z 1418.527,A 0.000,B 0.000,C 90.000,E1 310.782} C_DIS
LIN {X 0.262,Y -390.610,Z 1418.495,A 0.000,B 0.000,C 90.000,E1 305.025} C_DIS
LIN {X 0.106,Y -391.104,Z 1418.493,A 0.000,B 0.000,C 90.000,E1 304.692} C_DIS
LIN {X 0.022,Y -391.648,Z 1418.489,A 0.000,B 0.000,C 90.000,E1 303.992} C_DIS
LIN {X -0.080,Y -396.825,Z 1418.459,A 0.000,B 0.000,C 90.000,E1 298.693} C_DIS
LIN {X -0.210,Y -397.120,Z 1418.457,A 0.000,B 0.000,C 90.000,E1 298.359} C_DIS
LIN {X -0.055,Y -401.597,Z 1418.426,A 0.000,B 0.000,C 90.000,E1 292.717} C_DIS
LIN {X 0.222,Y -404.659,Z 1418.395,A 0.000,B 0.000,C 90.000,E1 287.094} C_DIS
LIN {X -0.079,Y -404.735,Z 1418.391,A 0.000,B 0.000,C 90.000,E1 286.441} C_DIS
LIN {X 0.214,Y -406.099,Z 1418.364,A 0.000,B 0.000,C 90.000,E1 281.535} C_DIS
LIN {X -0.176,Y -406.094,Z 1418.362,A 0.000,B 0.000,C 90.000,E1 281.243} C_DIS
LIN {X -0.097,Y -405.680,Z 1418.333,A 0.000,B 0.000,C 90.000,E1 276.024} C_DIS
LIN {X -0.165,Y -405.058,Z 1418.328,A 0.000,B 0.000,C 90.000,E1 274.992} C_DIS
LIN {X -0.060,Y -403.497,Z 1418.304,A 0.000,B 0.000,C 90.000,E1 270.802} C_DIS
LIN {X -0.092,Y -403.288,Z 1418.302,A 0.000,B 0.000,C 90.000,E1 270.458} C_DIS
LIN {X 0.091,Y -398.931,Z 1418.271,A 0.000,B 0.000,C 90.000,E1 264.837} C_DIS
LIN {X -0.040,Y -393.108,Z 1418.242,A 0.000,B 0.000,C 90.000,E1 259.567} C_DIS
LIN {X -0.079,Y -392.835,Z 1418.240,A 0.000,B 0.000,C 90.000,E1 259.218} C_DIS
LIN {X 0.034,Y -385.993,Z 1418.212,A 0.000,B 0.000,C 90.000,E1 254.212} C_DIS
LIN {X -0.026,Y -385.267,Z 1418.208,A 0.000,B 0.000,C 90.000,E1 253.504} C_DIS
LIN {X -0.004,Y -384.768,Z 1418.206,A 0.000,B 0.000,C 90.000,E1 253.142} C_DIS
LIN {X 0.221,Y -377.973,Z 1418.182,A 0.000,B 0.000,C 90.000,E1 248.773} C_DIS
LIN {X -0.044,Y -376.233,Z 1418.174,A 0.000,B 0.000,C 90.000,E1 247.358} C_DIS
LIN {X 0.057,Y -374.944,Z 1418.170,A 0.000,B 0.000,C 90.000,E1 246.613} C_DIS
LIN {X -0.208,Y -368.417,Z 1418.148,A 0.000,B 0.000,C 90.000,E1 242.615} C_DIS
LIN {X 0.097,Y -366.047,Z 1418.137,A 0.000,B 0.000,C 90.000,E1 240.717} C_DIS
LIN {X 0.004,Y -359.196,Z 1418.115,A 0.000,B 0.000,C 90.000,E1 236.628} C_DIS
LIN {X 0.021,Y -355.842,Z 1418.100,A 0.000,B 0.000,C 90.000,E1 233.989} C_DIS
LIN {X -0.173,Y -348.793,Z 1418.075,A 0.000,B 0.000,C 90.000,E1 229.461} C_DIS
LIN {X -0.097,Y -346.185,Z 1418.062,A 0.000,B 0.000,C 90.000,E1 227.148} C_DIS
LIN {X -0.088,Y -345.065,Z 1418.058,A 0.000,B 0.000,C 90.000,E1 226.377} C_DIS
LIN {X 0.094,Y -338.586,Z 1418.030,A 0.000,B 0.000,C 90.000,E1 221.310} C_DIS
LIN {X 0.094,Y -336.840,Z 1418.019,A 0.000,B 0.000,C 90.000,E1 219.358} C_DIS
LIN {X 0.014,Y -330.861,Z 1417.988,A 0.000,B 0.000,C 90.000,E1 213.865} C_DIS
LIN {X 0.149,Y -329.296,Z 1417.975,A 0.000,B 0.000,C 90.000,E1 211.465} C_DIS
LIN {X -0.154,Y -324.669,Z 1417.942,A 0.000,B 0.000,C 90.000,E1 205.540} C_DIS
LIN {X 0.174,Y -323.837,Z 1417.928,A 0.000,B 0.000,C 90.000,E1 203.078} C_DIS
LIN {X -0.017,Y -321.124,Z 1417.881,A 0.000,B 0.000,C 90.000,E1 194.662} C_DIS
LIN {X 0.138,Y -320.932,Z 1417.877,A 0.000,B 0.000,C 90.000,E1 193.828} C_DIS
LIN {X -0.076,Y -321.562,Z 1417.832,A 0.000,B 0.000,C 90.000,E1 185.796} C_DIS
LIN {X -0.143,Y -324.415,Z 1417.790,A 0.000,B 0.000,C 90.000,E1 178.165} C_DIS
LIN {X -0.141,Y -325.376,Z 1417.783,A 0.000,B 0.000,C 90.000,E1 176.963} C_DIS
LIN {X 0.050,Y -325.841,Z 1417.776,A 0.000,B 0.000,C 90.000,E1 175.698} C_DIS
LIN {X 0.030,Y -352.323,Z 1417.776,A 0.000,B 0.000,C 90.000,E1 175.698} C_DIS
LIN {X -0.113,Y -353.065,Z 1417.776,A 0.000,B 0.000,C 90.000,E1 175.698} C_DIS
LIN {X -0.102,Y -354.451,Z 1417.774,A 0.000,B 0.000,C 90.000,E1 175.355} C_DIS
LIN {X 0.050,Y -353.920,Z 1417.772,A 0.000,B 0.000,C 90.000,E1 174.951} C_DIS
LIN {X -0.177,Y -352.839,Z 1417.770,A 0.000,B 0.000,C 90.000,E1 174.609} C_DIS
LIN {X -0.140,Y -350.765,Z 1417.767,A 0.000,B 0.000,C 90.000,E1 174.033} C_DIS
LIN {X 0.018,Y -346.887,Z 1417.761,A 0.000,B 0.000,C 90.000,E1 173.053} C_DIS
LIN {X -0.005,Y -344.300,Z 1417.757,A 0.000,B 0.000,C 90.000,E1 172.299} C_DIS
LIN {X 0.112,Y -343.162,Z 1417.755,A 0.000,B 0.000,C 90.000,E1 171.894} C_DIS
LIN {X 0.140,Y -342.664,Z 1417.753,A 0.000,B 0.000,C 90.000,E1 171.546} C_DIS
LIN {X 0.122,Y -342.659,Z 1417.753,A 0.000,B 0.000,C 90.000,E1 171.546} C_DIS
LIN {X 0.093,Y -343.135,Z 1417.750,A 0.000,B 0.000,C 90.000,E1 171.027} C_DIS
LIN {X 0.070,Y -343.149,Z 1417.750,A 0.000,B 0.000,C 90.000,E1 170.971} C_DIS
LIN {X 0.051,Y -343.159,Z 1417.750,A 0.000,B 0.000,C 90.000,E1 170.971} C_DIS
LIN {X -0.128,Y -345.775,Z 1417.747,A 0.000,B 0.000,C 90.000,E1 170.387} C_DIS
LIN {X 0.139,Y -349.245,Z 1417.743,A 0.000,B 0.000,C 90.000,E1 169.746} C_DIS
LIN {X -0.018,Y -358.146,Z 1417.736,A 0.000,B 0.000,C 90.000,E1 168.522} C_DIS
LIN {X -0.013,Y -372.515,Z 1417.726,A 0.000,B 0.000,C 90.000,E1 166.700} C_DIS
LIN {X 0.080,Y -384.312,Z 1417.719,A 0.000,B 0.000,C 90.000,E1 165.338} C_DIS
LIN {X -0.084,Y -393.209,Z 1417.714,A 0.000,B 0.000,C 90.000,E1 164.448} C_DIS
LIN {X 0.125,Y -406.855,Z 1417.707,A 0.000,B 0.000,C 90.000,E1 163.142} C_DIS
LIN {X -0.195,Y -427.289,Z 1417.697,A 0.000,B 0.000,C 90.000,E1 161.456} C_DIS
LIN {X 0.238,Y -441.392,Z 1417.690,A 0.000,B 0.000,C 90.000,E1 160.242} C_DIS
LIN {X 0.071,Y -449.033,Z 1417.687,A 0.000,B 0.000,C 90.000,E1 159.625} C_DIS
LIN {X 0.142,Y -459.687,Z 1417.682,A 0.000,B 0.000,C 90.000,E1 158.720} C_DIS
LIN {X -0.040,Y -470.292,Z 1417.677,A 0.000,B 0.000,C 90.000,E1 157.847} C_DIS
LIN {X 0.107,Y -480.604,Z 1417.672,A 0.000,B 0.000,C 90.000,E1 156.922} C_DIS
LIN {X -0.219,Y -487.816,Z 1417.668,A 0.000,B 0.000,C 90.000,E1 156.305} C_DIS
LIN {X -0.101,Y -496.237,Z 1417.664,A 0.000,B 0.000,C 90.000,E1 155.485} C_DIS
LIN {X -0.044,Y -503.061,Z 1417.660,A 0.000,B 0.000,C 90.000,E1 154.793} C_DIS
LIN {X 0.033,Y -509.562,Z 1417.656,A 0.000,B 0.000,C 90.000,E1 154.076} C_DIS
LIN {X -0.141,Y -514.597,Z 1417.653,A 0.000,B 0.000,C 90.000,E1 153.512} C_DIS
LIN {X 0.031,Y -518.205,Z 1417.650,A 0.000,B 0.000,C 90.000,E1 153.050} C_DIS
LIN {X -0.174,Y -522.572,Z 1417.647,A 0.000,B 0.000,C 90.000,E1 152.487} C_DIS
LIN {X -0.108,Y -526.514,Z 1417.644,A 0.000,B 0.000,C 90.000,E1 151.897} C_DIS
LIN {X -0.011,Y -530.062,Z 1417.641,A 0.000,B 0.000,C 90.000,E1 151.307} C_DIS
LIN {X 0.115,Y -533.244,Z 1417.637,A 0.000,B 0.000,C 90.000,E1 150.717} C_DIS
LIN {X 0.265,Y -536.001,Z 1417.634,A 0.000,B 0.000,C 90.000,E1 150.127} C_DIS
LIN {X -0.031,Y -538.423,Z 1417.631,A 0.000,B 0.000,C 90.000,E1 149.587} C_DIS
LIN {X 0.155,Y -540.645,Z 1417.628,A 0.000,B 0.000,C 90.000,E1 148.997} C_DIS
LIN {X 0.079,Y -543.554,Z 1417.623,A 0.000,B 0.000,C 90.000,E1 148.152} C_DIS
LIN {X -0.145,Y -546.022,Z 1417.618,A 0.000,B 0.000,C 90.000,E1 147.327} C_DIS
LIN {X -0.338,Y -548.167,Z 1417.614,A 0.000,B 0.000,C 90.000,E1 146.501} C_DIS
LIN {X 0.254,Y -550.089,Z 1417.609,A 0.000,B 0.000,C 90.000,E1 145.595} C_DIS
LIN {X 0.103,Y -551.761,Z 1417.604,A 0.000,B 0.000,C 90.000,E1 144.769} C_DIS
LIN {X 0.289,Y -553.044,Z 1417.600,A 0.000,B 0.000,C 90.000,E1 143.909} C_DIS
LIN {X -0.282,Y -554.100,Z 1417.595,A 0.000,B 0.000,C 90.000,E1 143.130} C_DIS
LIN {X -0.069,Y -554.974,Z 1417.590,A 0.000,B 0.000,C 90.000,E1 142.271} C_DIS
LIN {X 0.016,Y -556.775,Z 1417.580,A 0.000,B 0.000,C 90.000,E1 140.312} C_DIS
LIN {X -0.170,Y -557.664,Z 1417.573,A 0.000,B 0.000,C 90.000,E1 139.218} C_DIS
LIN {X 0.162,Y -558.569,Z 1417.566,A 0.000,B 0.000,C 90.000,E1 137.796} C_DIS
LIN {X 0.131,Y -559.494,Z 1417.556,A 0.000,B 0.000,C 90.000,E1 136.134} C_DIS
LIN {X -0.278,Y -560.100,Z 1417.547,A 0.000,B 0.000,C 90.000,E1 134.514} C_DIS
LIN {X -0.273,Y -560.504,Z 1417.538,A 0.000,B 0.000,C 90.000,E1 132.852} C_DIS
LIN {X 0.063,Y -560.615,Z 1417.530,A 0.000,B 0.000,C 90.000,E1 131.434} C_DIS
LIN {X 0.107,Y -560.697,Z 1417.521,A 0.000,B 0.000,C 90.000,E1 129.769} C_DIS
LIN {X 0.232,Y -560.913,Z 1417.512,A 0.000,B 0.000,C 90.000,E1 128.096} C_DIS
LIN {X -0.070,Y -560.961,Z 1417.504,A 0.000,B 0.000,C 90.000,E1 126.744} C_DIS
LIN {X -0.272,Y -560.894,Z 1417.495,A 0.000,B 0.000,C 90.000,E1 125.105} C_DIS
LIN {X -0.119,Y -560.864,Z 1417.487,A 0.000,B 0.000,C 90.000,E1 123.706} C_DIS
LIN {X -0.155,Y -560.696,Z 1417.483,A 0.000,B 0.000,C 90.000,E1 122.880} C_DIS
LIN {X -0.059,Y -560.489,Z 1417.473,A 0.000,B 0.000,C 90.000,E1 121.209} C_DIS
LIN {X 0.043,Y -561.286,Z 1417.464,A 0.000,B 0.000,C 90.000,E1 119.539} C_DIS
LIN {X -0.093,Y -562.018,Z 1417.457,A 0.000,B 0.000,C 90.000,E1 118.309} C_DIS
LIN {X 0.175,Y -562.727,Z 1417.455,A 0.000,B 0.000,C 90.000,E1 117.897} C_DIS
LIN {X -0.119,Y -563.197,Z 1417.453,A 0.000,B 0.000,C 90.000,E1 117.513} C_DIS
LIN {X -0.037,Y -563.317,Z 1417.452,A 0.000,B 0.000,C 90.000,E1 117.436} C_DIS
LIN {X 0.189,Y -564.409,Z 1417.451,A 0.000,B 0.000,C 90.000,E1 117.206} C_DIS
LIN {X 0.094,Y -566.224,Z 1417.451,A 0.000,B 0.000,C 90.000,E1 117.078} C_DIS
LIN {X -0.182,Y -568.756,Z 1417.450,A 0.000,B 0.000,C 90.000,E1 117.001} C_DIS
LIN {X -0.110,Y -572.212,Z 1417.449,A 0.000,B 0.000,C 90.000,E1 116.796} C_DIS
LIN {X -0.015,Y -574.087,Z 1417.448,A 0.000,B 0.000,C 90.000,E1 116.693} C_DIS
LIN {X 0.064,Y -577.740,Z 1417.447,A 0.000,B 0.000,C 90.000,E1 116.411} C_DIS
LIN {X -0.011,Y -579.358,Z 1417.446,A 0.000,B 0.000,C 90.000,E1 116.309} C_DIS
LIN {X -0.033,Y -580.820,Z 1417.445,A 0.000,B 0.000,C 90.000,E1 116.104} C_DIS
LIN {X -0.174,Y -581.894,Z 1417.444,A 0.000,B 0.000,C 90.000,E1 115.848} C_DIS
LIN {X 0.215,Y -582.581,Z 1417.442,A 0.000,B 0.000,C 90.000,E1 115.540} C_DIS
LIN {X 0.083,Y -583.033,Z 1417.441,A 0.000,B 0.000,C 90.000,E1 115.283} C_DIS
LIN {X -0.046,Y -582.326,Z 1417.439,A 0.000,B 0.000,C 90.000,E1 115.027} C_DIS
LIN {X -0.243,Y -580.410,Z 1417.437,A 0.000,B 0.000,C 90.000,E1 114.643} C_DIS
LIN {X 0.219,Y -579.513,Z 1417.436,A 0.000,B 0.000,C 90.000,E1 114.463} C_DIS
LIN {X 0.232,Y -574.700,Z 1417.435,A 0.000,B 0.000,C 90.000,E1 114.259} C_DIS
LIN {X 0.214,Y -572.437,Z 1417.434,A 0.000,B 0.000,C 90.000,E1 114.079} C_DIS
LIN {X -0.172,Y -570.287,Z 1417.433,A 0.000,B 0.000,C 90.000,E1 114.003} C_DIS
LIN {X 0.007,Y -568.085,Z 1417.433,A 0.000,B 0.000,C 90.000,E1 113.898} C_DIS
LIN {X -0.187,Y -565.907,Z 1417.432,A 0.000,B 0.000,C 90.000,E1 113.770} C_DIS
LIN {X -0.042,Y -565.548,Z 1417.432,A 0.000,B 0.000,C 90.000,E1 113.695} C_DIS
LIN {X -0.136,Y -565.122,Z 1417.431,A 0.000,B 0.000,C 90.000,E1 113.567} C_DIS
LIN {X 0.097,Y -565.487,Z 1417.429,A 0.000,B 0.000,C 90.000,E1 113.131} C_DIS
LIN {X -0.220,Y -565.788,Z 1417.428,A 0.000,B 0.000,C 90.000,E1 113.025} C_DIS
LIN {X -0.126,Y -566.739,Z 1417.427,A 0.000,B 0.000,C 90.000,E1 112.770} C_DIS
LIN {X 0.134,Y -569.710,Z 1417.424,A 0.000,B 0.000,C 90.000,E1 112.386} C_DIS
LIN {X 0.106,Y -573.368,Z 1417.423,A 0.000,B 0.000,C 90.000,E1 112.153} C_DIS
LIN {X 0.243,Y -581.021,Z 1417.421,A 0.000,B 0.000,C 90.000,E1 111.770} C_DIS
LIN {X -0.102,Y -584.201,Z 1417.420,A 0.000,B 0.000,C 90.000,E1 111.642} C_DIS
LIN {X 0.020,Y -590.106,Z 1417.418,A 0.000,B 0.000,C 90.000,E1 111.280} C_DIS
LIN {X 0.206,Y -595.653,Z 1417.416,A 0.000,B 0.000,C 90.000,E1 110.865} C_DIS
LIN {X -0.014,Y -599.638,Z 1417.414,A 0.000,B 0.000,C 90.000,E1 110.556} C_DIS
LIN {X 0.095,Y -603.494,Z 1417.412,A 0.000,B 0.000,C 90.000,E1 110.194} C_DIS
LIN {X 0.153,Y -609.815,Z 1417.409,A 0.000,B 0.000,C 90.000,E1 109.577} C_DIS
LIN {X 0.015,Y -614.461,Z 1417.406,A 0.000,B 0.000,C 90.000,E1 109.087} C_DIS
LIN {X -0.264,Y -617.800,Z 1417.404,A 0.000,B 0.000,C 90.000,E1 108.725} C_DIS
LIN {X 0.046,Y -621.800,Z 1417.401,A 0.000,B 0.000,C 90.000,E1 108.181} C_DIS
LIN {X -0.209,Y -625.315,Z 1417.398,A 0.000,B 0.000,C 90.000,E1 107.692} C_DIS
LIN {X -0.034,Y -628.360,Z 1417.395,A 0.000,B 0.000,C 90.000,E1 107.166} C_DIS
LIN {X -0.251,Y -630.798,Z 1417.393,A 0.000,B 0.000,C 90.000,E1 106.677} C_DIS
LIN {X 0.159,Y -631.843,Z 1417.391,A 0.000,B 0.000,C 90.000,E1 106.386} C_DIS
LIN {X -0.046,Y -633.544,Z 1417.388,A 0.000,B 0.000,C 90.000,E1 105.898} C_DIS
LIN {X 0.198,Y -634.619,Z 1417.385,A 0.000,B 0.000,C 90.000,E1 105.371} C_DIS
LIN {X -0.173,Y -635.935,Z 1417.381,A 0.000,B 0.000,C 90.000,E1 104.647} C_DIS
LIN {X -0.082,Y -636.951,Z 1417.377,A 0.000,B 0.000,C 90.000,E1 103.883} C_DIS
LIN {X 0.195,Y -637.529,Z 1417.374,A 0.000,B 0.000,C 90.000,E1 103.355} C_DIS
LIN {X 0.307,Y -638.048,Z 1417.370,A 0.000,B 0.000,C 90.000,E1 102.591} C_DIS
LIN {X -0.031,Y -638.118,Z 1417.367,A 0.000,B 0.000,C 90.000,E1 102.119} C_DIS
LIN {X 0.253,Y -637.883,Z 1417.365,A 0.000,B 0.000,C 90.000,E1 101.591} C_DIS
LIN {X -0.214,Y -637.395,Z 1417.362,A 0.000,B 0.000,C 90.000,E1 101.130} C_DIS
LIN {X -0.109,Y -636.231,Z 1417.358,A 0.000,B 0.000,C 90.000,E1 100.366} C_DIS
LIN {X 0.049,Y -635.208,Z 1417.355,A 0.000,B 0.000,C 90.000,E1 99.849} C_DIS
LIN {X 0.309,Y -633.961,Z 1417.352,A 0.000,B 0.000,C 90.000,E1 99.321} C_DIS
LIN {X -0.169,Y -632.447,Z 1417.349,A 0.000,B 0.000,C 90.000,E1 98.859} C_DIS
LIN {X -0.226,Y -629.749,Z 1417.345,A 0.000,B 0.000,C 90.000,E1 98.106} C_DIS
LIN {X -0.099,Y -627.663,Z 1417.342,A 0.000,B 0.000,C 90.000,E1 97.587} C_DIS
LIN {X -0.060,Y -624.513,Z 1417.339,A 0.000,B 0.000,C 90.000,E1 96.947} C_DIS
LIN {X -0.126,Y -621.116,Z 1417.335,A 0.000,B 0.000,C 90.000,E1 96.315} C_DIS
LIN {X -0.218,Y -617.441,Z 1417.332,A 0.000,B 0.000,C 90.000,E1 95.682} C_DIS
LIN {X 0.141,Y -615.917,Z 1417.330,A 0.000,B 0.000,C 90.000,E1 95.391} C_DIS
LIN {X 0.002,Y -611.203,Z 1417.327,A 0.000,B 0.000,C 90.000,E1 94.759} C_DIS
LIN {X -0.052,Y -606.607,Z 1417.324,A 0.000,B 0.000,C 90.000,E1 94.245} C_DIS
LIN {X -0.003,Y -599.895,Z 1417.320,A 0.000,B 0.000,C 90.000,E1 93.612} C_DIS
LIN {X 0.085,Y -591.994,Z 1417.316,A 0.000,B 0.000,C 90.000,E1 92.922} C_DIS
LIN {X 0.036,Y -590.564,Z 1417.316,A 0.000,B 0.000,C 90.000,E1 92.808} C_DIS
LIN {X 0.174,Y -584.275,Z 1417.313,A 0.000,B 0.000,C 90.000,E1 92.350} C_DIS
LIN {X -0.251,Y -577.625,Z 1417.311,A 0.000,B 0.000,C 90.000,E1 92.007} C_DIS
LIN {X -0.137,Y -573.565,Z 1417.309,A 0.000,B 0.000,C 90.000,E1 91.661} C_DIS
LIN {X -0.174,Y -573.525,Z 1417.309,A 0.000,B 0.000,C 90.000,E1 91.661} C_DIS
LIN {X -0.101,Y -572.801,Z 1417.308,A 0.000,B 0.000,C 90.000,E1 91.432} C_DIS
LIN {X 0.086,Y -572.474,Z 1417.307,A 0.000,B 0.000,C 90.000,E1 91.146} C_DIS
LIN {X 0.008,Y -572.475,Z 1417.304,A 0.000,B 0.000,C 90.000,E1 90.745} C_DIS
LIN {X 0.136,Y -574.521,Z 1417.291,A 0.000,B 0.000,C 90.000,E1 88.282} C_DIS
LIN {X 0.164,Y -575.580,Z 1417.285,A 0.000,B 0.000,C 90.000,E1 87.192} C_DIS
LIN {X 0.115,Y -577.337,Z 1417.274,A 0.000,B 0.000,C 90.000,E1 85.298} C_DIS
LIN {X -0.141,Y -578.727,Z 1417.266,A 0.000,B 0.000,C 90.000,E1 83.970} C_DIS
LIN {X -0.214,Y -580.489,Z 1417.257,A 0.000,B 0.000,C 90.000,E1 82.356} C_DIS
LIN {X -0.202,Y -581.435,Z 1417.253,A 0.000,B 0.000,C 90.000,E1 81.546} C_DIS
LIN {X 0.080,Y -583.489,Z 1417.243,A 0.000,B 0.000,C 90.000,E1 79.634} C_DIS
LIN {X -0.194,Y -585.220,Z 1417.234,A 0.000,B 0.000,C 90.000,E1 78.049} C_DIS
LIN {X -0.104,Y -586.332,Z 1417.226,A 0.000,B 0.000,C 90.000,E1 76.700} C_DIS
LIN {X 0.141,Y -587.355,Z 1417.219,A 0.000,B 0.000,C 90.000,E1 75.338} C_DIS
LIN {X 0.088,Y -588.429,Z 1417.210,A 0.000,B 0.000,C 90.000,E1 73.740} C_DIS
LIN {X 0.206,Y -589.334,Z 1417.201,A 0.000,B 0.000,C 90.000,E1 72.127} C_DIS
LIN {X 0.070,Y -590.478,Z 1417.189,A 0.000,B 0.000,C 90.000,E1 70.007} C_DIS
LIN {X 0.166,Y -591.186,Z 1417.182,A 0.000,B 0.000,C 90.000,E1 68.666} C_DIS
LIN {X -0.164,Y -592.694,Z 1417.168,A 0.000,B 0.000,C 90.000,E1 66.305} C_DIS
LIN {X 0.046,Y -594.461,Z 1417.155,A 0.000,B 0.000,C 90.000,E1 63.896} C_DIS
LIN {X 0.124,Y -595.531,Z 1417.148,A 0.000,B 0.000,C 90.000,E1 62.564} C_DIS
LIN {X -0.127,Y -596.812,Z 1417.139,A 0.000,B 0.000,C 90.000,E1 61.001} C_DIS
LIN {X 0.164,Y -598.449,Z 1417.129,A 0.000,B 0.000,C 90.000,E1 59.125} C_DIS
LIN {X -0.088,Y -600.442,Z 1417.117,A 0.000,B 0.000,C 90.000,E1 57.041} C_DIS
LIN {X 0.364,Y -602.348,Z 1417.105,A 0.000,B 0.000,C 90.000,E1 54.895} C_DIS
LIN {X 0.209,Y -603.626,Z 1417.096,A 0.000,B 0.000,C 90.000,E1 53.336} C_DIS
LIN {X -0.191,Y -604.609,Z 1417.089,A 0.000,B 0.000,C 90.000,E1 52.065} C_DIS
LIN {X -0.038,Y -605.718,Z 1417.080,A 0.000,B 0.000,C 90.000,E1 50.481} C_DIS
LIN {X -0.305,Y -606.186,Z 1417.075,A 0.000,B 0.000,C 90.000,E1 49.461} C_DIS
LIN {X -0.181,Y -606.436,Z 1417.069,A 0.000,B 0.000,C 90.000,E1 48.405} C_DIS
LIN {X 0.218,Y -606.680,Z 1417.059,A 0.000,B 0.000,C 90.000,E1 46.539} C_DIS
LIN {X -0.353,Y -606.695,Z 1417.054,A 0.000,B 0.000,C 90.000,E1 45.810} C_DIS
LIN {X -0.017,Y -606.540,Z 1417.047,A 0.000,B 0.000,C 90.000,E1 44.474} C_DIS
LIN {X 0.093,Y -606.139,Z 1417.041,A 0.000,B 0.000,C 90.000,E1 43.419} C_DIS
LIN {X 0.179,Y -605.592,Z 1417.036,A 0.000,B 0.000,C 90.000,E1 42.366} C_DIS
LIN {X 0.092,Y -604.698,Z 1417.028,A 0.000,B 0.000,C 90.000,E1 41.067} C_DIS
LIN {X -0.060,Y -604.012,Z 1417.024,A 0.000,B 0.000,C 90.000,E1 40.297} C_DIS
LIN {X -0.316,Y -602.364,Z 1417.015,A 0.000,B 0.000,C 90.000,E1 38.749} C_DIS
LIN {X 0.215,Y -600.985,Z 1417.009,A 0.000,B 0.000,C 90.000,E1 37.649} C_DIS
LIN {X 0.115,Y -599.826,Z 1417.005,A 0.000,B 0.000,C 90.000,E1 36.870} C_DIS
LIN {X 0.247,Y -598.031,Z 1416.999,A 0.000,B 0.000,C 90.000,E1 35.804} C_DIS
LIN {X 0.009,Y -595.892,Z 1416.993,A 0.000,B 0.000,C 90.000,E1 34.771} C_DIS
LIN {X -0.139,Y -594.119,Z 1416.989,A 0.000,B 0.000,C 90.000,E1 33.992} C_DIS
LIN {X -0.219,Y -590.788,Z 1416.981,A 0.000,B 0.000,C 90.000,E1 32.673} C_DIS
LIN {X -0.252,Y -588.487,Z 1416.977,A 0.000,B 0.000,C 90.000,E1 31.878} C_DIS
LIN {X -0.123,Y -584.884,Z 1416.971,A 0.000,B 0.000,C 90.000,E1 30.797} C_DIS
LIN {X -0.210,Y -581.798,Z 1416.967,A 0.000,B 0.000,C 90.000,E1 30.001} C_DIS
LIN {X 0.034,Y -576.950,Z 1416.961,A 0.000,B 0.000,C 90.000,E1 28.899} C_DIS
LIN {X -0.141,Y -572.803,Z 1416.956,A 0.000,B 0.000,C 90.000,E1 28.103} C_DIS
LIN {X 0.138,Y -568.373,Z 1416.952,A 0.000,B 0.000,C 90.000,E1 27.257} C_DIS
LIN {X 0.111,Y -563.613,Z 1416.947,A 0.000,B 0.000,C 90.000,E1 26.437} C_DIS
LIN {X -0.123,Y -559.313,Z 1416.943,A 0.000,B 0.000,C 90.000,E1 25.771} C_DIS
LIN {X 0.259,Y -553.806,Z 1416.938,A 0.000,B 0.000,C 90.000,E1 24.899} C_DIS
LIN {X -0.188,Y -549.874,Z 1416.935,A 0.000,B 0.000,C 90.000,E1 24.387} C_DIS
LIN {X 0.217,Y -544.542,Z 1416.932,A 0.000,B 0.000,C 90.000,E1 23.643} C_DIS
LIN {X 0.206,Y -540.011,Z 1416.928,A 0.000,B 0.000,C 90.000,E1 23.078} C_DIS
LIN {X 0.159,Y -535.173,Z 1416.925,A 0.000,B 0.000,C 90.000,E1 22.514} C_DIS
LIN {X -0.210,Y -527.957,Z 1416.921,A 0.000,B 0.000,C 90.000,E1 21.716} C_DIS
LIN {X 0.213,Y -522.719,Z 1416.917,A 0.000,B 0.000,C 90.000,E1 21.099} C_DIS
LIN {X -0.161,Y -514.880,Z 1416.913,A 0.000,B 0.000,C 90.000,E1 20.301} C_DIS
LIN {X -0.135,Y -504.324,Z 1416.907,A 0.000,B 0.000,C 90.000,E1 19.214} C_DIS
LIN {X 0.214,Y -495.130,Z 1416.901,A 0.000,B 0.000,C 90.000,E1 18.236} C_DIS
LIN {X -0.050,Y -480.350,Z 1416.893,A 0.000,B 0.000,C 90.000,E1 16.732} C_DIS
LIN {X 0.261,Y -466.914,Z 1416.885,A 0.000,B 0.000,C 90.000,E1 15.245} C_DIS
LIN {X -0.179,Y -454.647,Z 1416.877,A 0.000,B 0.000,C 90.000,E1 13.939} C_DIS
LIN {X -0.053,Y -441.228,Z 1416.869,A 0.000,B 0.000,C 90.000,E1 12.411} C_DIS
LIN {X 0.016,Y -422.316,Z 1416.856,A 0.000,B 0.000,C 90.000,E1 10.141} C_DIS
LIN {X -0.028,Y -404.018,Z 1416.843,A 0.000,B 0.000,C 90.000,E1 7.757} C_DIS
LIN {X -0.057,Y -397.615,Z 1416.838,A 0.000,B 0.000,C 90.000,E1 6.891} C_DIS
LIN {X 0.194,Y -389.382,Z 1416.832,A 0.000,B 0.000,C 90.000,E1 5.796} C_DIS
LIN {X 0.154,Y -387.967,Z 1416.831,A 0.000,B 0.000,C 90.000,E1 5.625} C_DIS
LIN {X -0.030,Y -383.902,Z 1416.828,A 0.000,B 0.000,C 90.000,E1 5.049} C_DIS
LIN {X 0.135,Y -383.453,Z 1416.828,A 0.000,B 0.000,C 90.000,E1 4.935} C_DIS
LIN {X 0.142,Y -382.709,Z 1416.826,A 0.000,B 0.000,C 90.000,E1 4.702} C_DIS
LIN {X 0.110,Y -382.708,Z 1416.826,A 0.000,B 0.000,C 90.000,E1 4.702} C_DIS
LIN {X 0.086,Y -383.562,Z 1416.823,A 0.000,B 0.000,C 90.000,E1 4.188} C_DIS
LIN {X -0.005,Y -383.800,Z 1416.821,A 0.000,B 0.000,C 90.000,E1 3.841} C_DIS
LIN {X -0.094,Y -383.518,Z 1416.820,A 0.000,B 0.000,C 90.000,E1 3.669} C_DIS
LIN {X 0.065,Y -382.860,Z 1416.820,A 0.000,B 0.000,C 90.000,E1 3.555} C_DIS
LIN {X 0.113,Y -381.726,Z 1416.820,A 0.000,B 0.000,C 90.000,E1 3.498} C_DIS
LIN {X 0.070,Y -361.596,Z 1416.820,A 0.000,B 0.000,C 90.000,E1 3.498} C_DIS
LIN {X -0.033,Y -360.861,Z 1416.801,A 0.000,B 0.000,C 90.000,E1 0.115} C_DIS
LIN {X -0.053,Y -359.426,Z 1416.770,A 0.000,B 0.000,C 90.000,E1 354.546} C_DIS
LIN {X 0.070,Y -358.890,Z 1416.759,A 0.000,B 0.000,C 90.000,E1 352.648} C_DIS
LIN {X -0.020,Y -359.563,Z 1416.726,A 0.000,B 0.000,C 90.000,E1 346.645} C_DIS
LIN {X 0.001,Y -361.801,Z 1416.684,A 0.000,B 0.000,C 90.000,E1 339.135} C_DIS
LIN {X -0.154,Y -362.053,Z 1416.680,A 0.000,B 0.000,C 90.000,E1 338.411} C_DIS
LIN {X 0.189,Y -365.980,Z 1416.643,A 0.000,B 0.000,C 90.000,E1 331.641} C_DIS
LIN {X 0.029,Y -366.387,Z 1416.639,A 0.000,B 0.000,C 90.000,E1 330.923} C_DIS
LIN {X -0.031,Y -371.355,Z 1416.604,A 0.000,B 0.000,C 90.000,E1 324.642} C_DIS
LIN {X -0.043,Y -371.766,Z 1416.602,A 0.000,B 0.000,C 90.000,E1 324.276} C_DIS
LIN {X 0.013,Y -377.358,Z 1416.567,A 0.000,B 0.000,C 90.000,E1 318.038} C_DIS
LIN {X 0.012,Y -378.235,Z 1416.563,A 0.000,B 0.000,C 90.000,E1 317.310} C_DIS
LIN {X 0.002,Y -383.940,Z 1416.531,A 0.000,B 0.000,C 90.000,E1 311.515} C_DIS
LIN {X 0.088,Y -384.893,Z 1416.527,A 0.000,B 0.000,C 90.000,E1 310.782} C_DIS
LIN {X 0.262,Y -390.610,Z 1416.495,A 0.000,B 0.000,C 90.000,E1 305.025} C_DIS
LIN {X 0.106,Y -391.104,Z 1416.493,A 0.000,B 0.000,C 90.000,E1 304.692} C_DIS
LIN {X 0.022,Y -391.648,Z 1416.489,A 0.000,B 0.000,C 90.000,E1 303.992} C_DIS
LIN {X -0.080,Y -396.825,Z 1416.459,A 0.000,B 0.000,C 90.000,E1 298.693} C_DIS
LIN {X -0.210,Y -397.120,Z 1416.457,A 0.000,B 0.000,C 90.000,E1 298.359} C_DIS
LIN {X -0.055,Y -401.597,Z 1416.426,A 0.000,B 0.000,C 90.000,E1 292.717} C_DIS
LIN {X 0.222,Y -404.659,Z 1416.395,A 0.000,B 0.000,C 90.000,E1 287.094} C_DIS
LIN {X -0.079,Y -404.735,Z 1416.391,A 0.000,B 0.000,C 90.000,E1 286.441} C_DIS
LIN {X 0.214,Y -406.099,Z 1416.364,A 0.000,B 0.000,C 90.000,E1 281.535} C_DIS
LIN {X -0.176,Y -406.094,Z 1416.362,A 0.000,B 0.000,C 90.000,E1 281.243} C_DIS
LIN {X -0.097,Y -405.680,Z 1416.333,A 0.000,B 0.000,C 90.000,E1 276.024} C_DIS
LIN {X -0.165,Y -405.058,Z 1416.328,A 0.000,B 0.000,C 90.000,E1 274.992} C_DIS
LIN {X -0.060,Y -403.497,Z 1416.304,A 0.000,B 0.000,C 90.000,E1 270.802} C_DIS
LIN {X -0.092,Y -403.288,Z 1416.302,A 0.000,B 0.000,C 90.000,E1 270.458} C_DIS
LIN {X 0.091,Y -398.931,Z 1416.271,A 0.000,B 0.000,C 90.000,E1 264.837} C_DIS
LIN {X -0.040,Y -393.108,Z 1416.242,A 0.000,B 0.000,C 90.000,E1 259.567} C_DIS
LIN {X -0.079,Y -392.835,Z 1416.240,A 0.000,B 0.000,C 90.000,E1 259.218} C_DIS
LIN {X 0.034,Y -385.993,Z 1416.212,A 0.000,B 0.000,C 90.000,E1 254.212} C_DIS
LIN {X -0.026,Y -385.267,Z 1416.208,A 0.000,B 0.000,C 90.000,E1 253.504} C_DIS
LIN {X -0.004,Y -384.768,Z 1416.206,A 0.000,B 0.000,C 90.000,E1 253.142} C_DIS
LIN {X 0.221,Y -377.973,Z 1416.182,A 0.000,B 0.000,C 90.000,E1 248.773} C_DIS
LIN {X -0.044,Y -376.233,Z 1416.174,A 0.000,B 0.000,C 90.000,E1 247.358} C_DIS
LIN {X 0.057,Y -374.944,Z 1416.170,A 0.000,B 0.000,C 90.000,E1 246.613} C_DIS
LIN {X -0.208,Y -368.417,Z 1416.148,A 0.000,B 0.000,C 90.000,E1 242.615} C_DIS
LIN {X 0.097,Y -366.047,Z 1416.137,A 0.000,B 0.000,C 90.000,E1 240.717} C_DIS
LIN {X 0.004,Y -359.196,Z 1416.115,A 0.000,B 0.000,C 90.000,E1 236.628} C_DIS
LIN {X 0.021,Y -355.842,Z 1416.100,A 0.000,B 0.000,C 90.000,E1 233.989} C_DIS
LIN {X -0.173,Y -348.793,Z 1416.075,A 0.000,B 0.000,C 90.000,E1 229.461} C_DIS
LIN {X -0.097,Y -346.185,Z 1416.062,A 0.000,B 0.000,C 90.000,E1 227.148} C_DIS
LIN {X -0.088,Y -345.065,Z 1416.058,A 0.000,B 0.000,C 90.000,E1 226.377} C_DIS
LIN {X 0.094,Y -338.586,Z 1416.030,A 0.000,B 0.000,C 90.000,E1 221.310} C_DIS
LIN {X 0.094,Y -336.840,Z 1416.019,A 0.000,B 0.000,C 90.000,E1 219.358} C_DIS
LIN {X 0.014,Y -330.861,Z 1415.988,A 0.000,B 0.000,C 90.000,E1 213.865} C_DIS
LIN {X 0.149,Y -329.296,Z 1415.975,A 0.000,B 0.000,C 90.000,E1 211.465} C_DIS
LIN {X -0.154,Y -324.669,Z 1415.942,A 0.000,B 0.000,C 90.000,E1 205.540} C_DIS
LIN {X 0.174,Y -323.837,Z 1415.928,A 0.000,B 0.000,C 90.000,E1 203.078} C_DIS
LIN {X -0.017,Y -321.124,Z 1415.881,A 0.000,B 0.000,C 90.000,E1 194.662} C_DIS
LIN {X 0.138,Y -320.932,Z 1415.877,A 0.000,B 0.000,C 90.000,E1 193.828} C_DIS
LIN {X -0.076,Y -321.562,Z 1415.832,A 0.000,B 0.000,C 90.000,E1 185.796} C_DIS
LIN {X -0.143,Y -324.415,Z 1415.790,A 0.000,B 0.000,C 90.000,E1 178.165} C_DIS
LIN {X -0.136,Y -325.416,Z 1415.782,A 0.000,B 0.000,C 90.000,E1 176.846} C_DIS
LIN {X 0.186,Y -360.469,Z 1415.782,A 0.000,B 0.000,C 90.000,E1 176.788} C_DIS
LIN {X 0.049,Y -361.544,Z 1415.782,A 0.000,B 0.000,C 90.000,E1 176.788} C_DIS
LIN {X -0.135,Y -363.015,Z 1415.781,A 0.000,B 0.000,C 90.000,E1 176.560} C_DIS
LIN {X 0.029,Y -362.550,Z 1415.779,A 0.000,B 0.000,C 90.000,E1 176.159} C_DIS
LIN {X 0.126,Y -360.752,Z 1415.776,A 0.000,B 0.000,C 90.000,E1 175.584} C_DIS
LIN {X -0.143,Y -358.409,Z 1415.772,A 0.000,B 0.000,C 90.000,E1 175.065} C_DIS
LIN {X 0.177,Y -349.197,Z 1415.761,A 0.000,B 0.000,C 90.000,E1 172.932} C_DIS
LIN {X -0.154,Y -347.045,Z 1415.758,A 0.000,B 0.000,C 90.000,E1 172.413} C_DIS
LIN {X -0.031,Y -344.224,Z 1415.752,A 0.000,B 0.000,C 90.000,E1 171.432} C_DIS
LIN {X 0.086,Y -344.007,Z 1415.750,A 0.000,B 0.000,C 90.000,E1 171.027} C_DIS
LIN {X 0.081,Y -343.993,Z 1415.750,A 0.000,B 0.000,C 90.000,E1 170.971} C_DIS
LIN {X 0.064,Y -343.998,Z 1415.750,A 0.000,B 0.000,C 90.000,E1 170.971} C_DIS
LIN {X 0.115,Y -345.692,Z 1415.747,A 0.000,B 0.000,C 90.000,E1 170.443} C_DIS
LIN {X 0.018,Y -349.927,Z 1415.743,A 0.000,B 0.000,C 90.000,E1 169.690} C_DIS
LIN {X 0.137,Y -357.658,Z 1415.737,A 0.000,B 0.000,C 90.000,E1 168.578} C_DIS
LIN {X 0.027,Y -369.169,Z 1415.729,A 0.000,B 0.000,C 90.000,E1 167.117} C_DIS
LIN {X -0.089,Y -380.916,Z 1415.721,A 0.000,B 0.000,C 90.000,E1 165.755} C_DIS
LIN {X 0.032,Y -391.357,Z 1415.715,A 0.000,B 0.000,C 90.000,E1 164.629} C_DIS
LIN {X 0.106,Y -405.011,Z 1415.708,A 0.000,B 0.000,C 90.000,E1 163.323} C_DIS
LIN {X 0.129,Y -427.001,Z 1415.697,A 0.000,B 0.000,C 90.000,E1 161.456} C_DIS
LIN {X 0.056,Y -441.062,Z 1415.691,A 0.000,B 0.000,C 90.000,E1 160.315} C_DIS
LIN {X -0.139,Y -450.299,Z 1415.686,A 0.000,B 0.000,C 90.000,E1 159.571} C_DIS
LIN {X 0.184,Y -460.820,Z 1415.682,A 0.000,B 0.000,C 90.000,E1 158.646} C_DIS
LIN {X -0.165,Y -471.380,Z 1415.677,A 0.000,B 0.000,C 90.000,E1 157.794} C_DIS
LIN {X -0.101,Y -481.746,Z 1415.672,A 0.000,B 0.000,C 90.000,E1 156.869} C_DIS
LIN {X 0.192,Y -488.914,Z 1415.668,A 0.000,B 0.000,C 90.000,E1 156.177} C_DIS
LIN {X -0.193,Y -497.401,Z 1415.663,A 0.000,B 0.000,C 90.000,E1 155.409} C_DIS
LIN {X -0.183,Y -504.123,Z 1415.659,A 0.000,B 0.000,C 90.000,E1 154.717} C_DIS
LIN {X -0.236,Y -509.363,Z 1415.656,A 0.000,B 0.000,C 90.000,E1 154.152} C_DIS
LIN {X 0.285,Y -514.407,Z 1415.653,A 0.000,B 0.000,C 90.000,E1 153.512} C_DIS
LIN {X -0.232,Y -518.006,Z 1415.651,A 0.000,B 0.000,C 90.000,E1 153.127} C_DIS
LIN {X 0.261,Y -522.438,Z 1415.647,A 0.000,B 0.000,C 90.000,E1 152.487} C_DIS
LIN {X 0.329,Y -526.444,Z 1415.644,A 0.000,B 0.000,C 90.000,E1 151.897} C_DIS
LIN {X -0.291,Y -530.017,Z 1415.641,A 0.000,B 0.000,C 90.000,E1 151.385} C_DIS
LIN {X -0.169,Y -533.228,Z 1415.638,A 0.000,B 0.000,C 90.000,E1 150.795} C_DIS
LIN {X -0.166,Y -536.608,Z 1415.634,A 0.000,B 0.000,C 90.000,E1 150.078} C_DIS
LIN {X 0.138,Y -539.559,Z 1415.630,A 0.000,B 0.000,C 90.000,E1 149.331} C_DIS
LIN {X -0.136,Y -541.674,Z 1415.627,A 0.000,B 0.000,C 90.000,E1 148.791} C_DIS
LIN {X 0.068,Y -543.572,Z 1415.623,A 0.000,B 0.000,C 90.000,E1 148.201} C_DIS
LIN {X -0.153,Y -546.051,Z 1415.619,A 0.000,B 0.000,C 90.000,E1 147.375} C_DIS
LIN {X 0.115,Y -548.206,Z 1415.614,A 0.000,B 0.000,C 90.000,E1 146.501} C_DIS
LIN {X -0.055,Y -550.113,Z 1415.609,A 0.000,B 0.000,C 90.000,E1 145.674} C_DIS
LIN {X 0.111,Y -551.767,Z 1415.605,A 0.000,B 0.000,C 90.000,E1 144.815} C_DIS
LIN {X -0.024,Y -553.039,Z 1415.600,A 0.000,B 0.000,C 90.000,E1 143.989} C_DIS
LIN {X 0.178,Y -554.087,Z 1415.595,A 0.000,B 0.000,C 90.000,E1 143.130} C_DIS
LIN {X -0.048,Y -554.932,Z 1415.591,A 0.000,B 0.000,C 90.000,E1 142.316} C_DIS
LIN {X 0.048,Y -556.728,Z 1415.580,A 0.000,B 0.000,C 90.000,E1 140.356} C_DIS
LIN {X -0.073,Y -557.616,Z 1415.574,A 0.000,B 0.000,C 90.000,E1 139.256} C_DIS
LIN {X -0.240,Y -558.340,Z 1415.568,A 0.000,B 0.000,C 90.000,E1 138.162} C_DIS
LIN {X -0.199,Y -559.422,Z 1415.557,A 0.000,B 0.000,C 90.000,E1 136.215} C_DIS
LIN {X 0.182,Y -560.026,Z 1415.547,A 0.000,B 0.000,C 90.000,E1 134.514} C_DIS
LIN {X 0.185,Y -560.434,Z 1415.538,A 0.000,B 0.000,C 90.000,E1 132.852} C_DIS
LIN {X 0.148,Y -560.554,Z 1415.531,A 0.000,B 0.000,C 90.000,E1 131.472} C_DIS
LIN {X 0.204,Y -560.635,Z 1415.521,A 0.000,B 0.000,C 90.000,E1 129.806} C_DIS
LIN {X -0.101,Y -560.880,Z 1415.512,A 0.000,B 0.000,C 90.000,E1 128.177} C_DIS
LIN {X -0.065,Y -560.939,Z 1415.504,A 0.000,B 0.000,C 90.000,E1 126.790} C_DIS
LIN {X 0.182,Y -560.893,Z 1415.495,A 0.000,B 0.000,C 90.000,E1 125.105} C_DIS
LIN {X 0.334,Y -560.866,Z 1415.488,A 0.000,B 0.000,C 90.000,E1 123.706} C_DIS
LIN {X 0.083,Y -560.663,Z 1415.481,A 0.000,B 0.000,C 90.000,E1 122.625} C_DIS
LIN {X -0.293,Y -560.757,Z 1415.472,A 0.000,B 0.000,C 90.000,E1 121.003} C_DIS
LIN {X 0.015,Y -561.682,Z 1415.464,A 0.000,B 0.000,C 90.000,E1 119.589} C_DIS
LIN {X 0.177,Y -562.250,Z 1415.460,A 0.000,B 0.000,C 90.000,E1 118.743} C_DIS
LIN {X -0.022,Y -562.478,Z 1415.458,A 0.000,B 0.000,C 90.000,E1 118.487} C_DIS
LIN {X 0.192,Y -563.583,Z 1415.456,A 0.000,B 0.000,C 90.000,E1 118.025} C_DIS
LIN {X 0.149,Y -563.624,Z 1415.456,A 0.000,B 0.000,C 90.000,E1 118.025} C_DIS
LIN {X 0.085,Y -564.653,Z 1415.455,A 0.000,B 0.000,C 90.000,E1 117.924} C_DIS
LIN {X 0.251,Y -565.578,Z 1415.455,A 0.000,B 0.000,C 90.000,E1 117.847} C_DIS
LIN {X -0.350,Y -567.158,Z 1415.455,A 0.000,B 0.000,C 90.000,E1 117.847} C_DIS
LIN {X 0.250,Y -572.194,Z 1415.454,A 0.000,B 0.000,C 90.000,E1 117.641} C_DIS
LIN {X -0.238,Y -575.955,Z 1415.453,A 0.000,B 0.000,C 90.000,E1 117.513} C_DIS
LIN {X 0.273,Y -577.738,Z 1415.452,A 0.000,B 0.000,C 90.000,E1 117.385} C_DIS
LIN {X 0.118,Y -583.035,Z 1415.450,A 0.000,B 0.000,C 90.000,E1 117.052} C_DIS
LIN {X -0.164,Y -585.816,Z 1415.448,A 0.000,B 0.000,C 90.000,E1 116.744} C_DIS
LIN {X -0.290,Y -587.972,Z 1415.447,A 0.000,B 0.000,C 90.000,E1 116.488} C_DIS
LIN {X 0.177,Y -588.700,Z 1415.446,A 0.000,B 0.000,C 90.000,E1 116.309} C_DIS
LIN {X -0.043,Y -590.565,Z 1415.443,A 0.000,B 0.000,C 90.000,E1 115.796} C_DIS
LIN {X -0.149,Y -591.235,Z 1415.442,A 0.000,B 0.000,C 90.000,E1 115.540} C_DIS
LIN {X -0.353,Y -590.191,Z 1415.439,A 0.000,B 0.000,C 90.000,E1 115.027} C_DIS
LIN {X 0.078,Y -589.191,Z 1415.437,A 0.000,B 0.000,C 90.000,E1 114.719} C_DIS
LIN {X -0.083,Y -585.950,Z 1415.435,A 0.000,B 0.000,C 90.000,E1 114.335} C_DIS
LIN {X -0.140,Y -584.641,Z 1415.434,A 0.000,B 0.000,C 90.000,E1 114.207} C_DIS
LIN {X -0.189,Y -569.679,Z 1415.430,A 0.000,B 0.000,C 90.000,E1 113.462} C_DIS
LIN {X 0.227,Y -567.490,Z 1415.429,A 0.000,B 0.000,C 90.000,E1 113.259} C_DIS
LIN {X 0.192,Y -567.447,Z 1415.429,A 0.000,B 0.000,C 90.000,E1 113.259} C_DIS
LIN {X 0.074,Y -567.706,Z 1415.428,A 0.000,B 0.000,C 90.000,E1 112.950} C_DIS
LIN {X 0.061,Y -569.845,Z 1415.426,A 0.000,B 0.000,C 90.000,E1 112.695} C_DIS
LIN {X -0.250,Y -571.137,Z 1415.425,A 0.000,B 0.000,C 90.000,E1 112.589} C_DIS
LIN {X -0.083,Y -574.670,Z 1415.424,A 0.000,B 0.000,C 90.000,E1 112.333} C_DIS
LIN {X 0.192,Y -585.247,Z 1415.421,A 0.000,B 0.000,C 90.000,E1 111.770} C_DIS
LIN {X 0.261,Y -591.154,Z 1415.419,A 0.000,B 0.000,C 90.000,E1 111.408} C_DIS
LIN {X -0.149,Y -596.723,Z 1415.417,A 0.000,B 0.000,C 90.000,E1 111.046} C_DIS
LIN {X -0.040,Y -602.108,Z 1415.415,A 0.000,B 0.000,C 90.000,E1 110.610} C_DIS
LIN {X 0.203,Y -608.387,Z 1415.411,A 0.000,B 0.000,C 90.000,E1 109.993} C_DIS
LIN {X 0.055,Y -613.434,Z 1415.408,A 0.000,B 0.000,C 90.000,E1 109.504} C_DIS
LIN {X -0.180,Y -617.893,Z 1415.406,A 0.000,B 0.000,C 90.000,E1 109.014} C_DIS
LIN {X -0.324,Y -621.881,Z 1415.403,A 0.000,B 0.000,C 90.000,E1 108.544} C_DIS
LIN {X 0.177,Y -626.404,Z 1415.399,A 0.000,B 0.000,C 90.000,E1 107.873} C_DIS
LIN {X -0.167,Y -630.940,Z 1415.395,A 0.000,B 0.000,C 90.000,E1 107.149} C_DIS
LIN {X -0.139,Y -634.230,Z 1415.391,A 0.000,B 0.000,C 90.000,E1 106.386} C_DIS
LIN {X 0.283,Y -635.667,Z 1415.388,A 0.000,B 0.000,C 90.000,E1 105.843} C_DIS
LIN {X -0.070,Y -636.766,Z 1415.385,A 0.000,B 0.000,C 90.000,E1 105.371} C_DIS
LIN {X 0.195,Y -637.973,Z 1415.381,A 0.000,B 0.000,C 90.000,E1 104.592} C_DIS
LIN {X -0.020,Y -639.592,Z 1415.374,A 0.000,B 0.000,C 90.000,E1 103.355} C_DIS
LIN {X 0.113,Y -639.969,Z 1415.370,A 0.000,B 0.000,C 90.000,E1 102.591} C_DIS
LIN {X -0.213,Y -640.048,Z 1415.367,A 0.000,B 0.000,C 90.000,E1 102.119} C_DIS
LIN {X 0.086,Y -639.784,Z 1415.365,A 0.000,B 0.000,C 90.000,E1 101.591} C_DIS
LIN {X 0.091,Y -638.976,Z 1415.360,A 0.000,B 0.000,C 90.000,E1 100.838} C_DIS
LIN {X -0.246,Y -638.159,Z 1415.358,A 0.000,B 0.000,C 90.000,E1 100.366} C_DIS
LIN {X -0.074,Y -637.148,Z 1415.355,A 0.000,B 0.000,C 90.000,E1 99.849} C_DIS
LIN {X 0.199,Y -635.899,Z 1415.352,A 0.000,B 0.000,C 90.000,E1 99.321} C_DIS
LIN {X -0.266,Y -634.372,Z 1415.349,A 0.000,B 0.000,C 90.000,E1 98.859} C_DIS
LIN {X -0.110,Y -632.611,Z 1415.346,A 0.000,B 0.000,C 90.000,E1 98.341} C_DIS
LIN {X -0.164,Y -629.537,Z 1415.342,A 0.000,B 0.000,C 90.000,E1 97.587} C_DIS
LIN {X -0.106,Y -626.512,Z 1415.339,A 0.000,B 0.000,C 90.000,E1 96.947} C_DIS
LIN {X -0.153,Y -623.065,Z 1415.335,A 0.000,B 0.000,C 90.000,E1 96.315} C_DIS
LIN {X 0.234,Y -618.704,Z 1415.331,A 0.000,B 0.000,C 90.000,E1 95.511} C_DIS
LIN {X -0.018,Y -617.052,Z 1415.329,A 0.000,B 0.000,C 90.000,E1 95.277} C_DIS
LIN {X 0.015,Y -613.346,Z 1415.327,A 0.000,B 0.000,C 90.000,E1 94.759} C_DIS
LIN {X 0.138,Y -610.081,Z 1415.324,A 0.000,B 0.000,C 90.000,E1 94.359} C_DIS
LIN {X -0.190,Y -607.634,Z 1415.323,A 0.000,B 0.000,C 90.000,E1 94.131} C_DIS
LIN {X 0.114,Y -602.512,Z 1415.320,A 0.000,B 0.000,C 90.000,E1 93.612} C_DIS
LIN {X 0.205,Y -596.032,Z 1415.317,A 0.000,B 0.000,C 90.000,E1 93.037} C_DIS
LIN {X 0.043,Y -590.280,Z 1415.314,A 0.000,B 0.000,C 90.000,E1 92.579} C_DIS
LIN {X -0.284,Y -583.867,Z 1415.312,A 0.000,B 0.000,C 90.000,E1 92.178} C_DIS
LIN {X -0.061,Y -577.269,Z 1415.310,A 0.000,B 0.000,C 90.000,E1 91.776} C_DIS
LIN {X -0.256,Y -573.676,Z 1415.308,A 0.000,B 0.000,C 90.000,E1 91.489} C_DIS
LIN {X 0.281,Y -573.658,Z 1415.308,A 0.000,B 0.000,C 90.000,E1 91.432} C_DIS
LIN {X -0.266,Y -573.021,Z 1415.307,A 0.000,B 0.000,C 90.000,E1 91.318} C_DIS
LIN {X -0.233,Y -572.611,Z 1415.306,A 0.000,B 0.000,C 90.000,E1 91.031} C_DIS
LIN {X 0.047,Y -572.665,Z 1415.303,A 0.000,B 0.000,C 90.000,E1 90.458} C_DIS
LIN {X -0.108,Y -574.261,Z 1415.292,A 0.000,B 0.000,C 90.000,E1 88.568} C_DIS
LIN {X 0.062,Y -575.571,Z 1415.284,A 0.000,B 0.000,C 90.000,E1 87.192} C_DIS
LIN {X 0.013,Y -577.316,Z 1415.274,A 0.000,B 0.000,C 90.000,E1 85.298} C_DIS
LIN {X -0.244,Y -578.736,Z 1415.266,A 0.000,B 0.000,C 90.000,E1 83.970} C_DIS
LIN {X 0.258,Y -580.504,Z 1415.257,A 0.000,B 0.000,C 90.000,E1 82.299} C_DIS
LIN {X -0.077,Y -581.731,Z 1415.251,A 0.000,B 0.000,C 90.000,E1 81.254} C_DIS
LIN {X -0.023,Y -583.533,Z 1415.242,A 0.000,B 0.000,C 90.000,E1 79.634} C_DIS
LIN {X 0.276,Y -585.243,Z 1415.234,A 0.000,B 0.000,C 90.000,E1 77.993} C_DIS
LIN {X -0.207,Y -586.346,Z 1415.226,A 0.000,B 0.000,C 90.000,E1 76.700} C_DIS
LIN {X 0.212,Y -587.212,Z 1415.220,A 0.000,B 0.000,C 90.000,E1 75.589} C_DIS
LIN {X 0.304,Y -588.273,Z 1415.211,A 0.000,B 0.000,C 90.000,E1 73.976} C_DIS
LIN {X 0.006,Y -589.023,Z 1415.204,A 0.000,B 0.000,C 90.000,E1 72.670} C_DIS
LIN {X 0.208,Y -589.609,Z 1415.198,A 0.000,B 0.000,C 90.000,E1 71.583} C_DIS
LIN {X 0.283,Y -590.807,Z 1415.186,A 0.000,B 0.000,C 90.000,E1 69.444} C_DIS
LIN {X -0.052,Y -591.845,Z 1415.176,A 0.000,B 0.000,C 90.000,E1 67.614} C_DIS
LIN {X 0.077,Y -593.107,Z 1415.165,A 0.000,B 0.000,C 90.000,E1 65.741} C_DIS
LIN {X -0.053,Y -594.507,Z 1415.155,A 0.000,B 0.000,C 90.000,E1 63.896} C_DIS
LIN {X 0.025,Y -595.575,Z 1415.148,A 0.000,B 0.000,C 90.000,E1 62.564} C_DIS
LIN {X 0.065,Y -596.855,Z 1415.139,A 0.000,B 0.000,C 90.000,E1 60.973} C_DIS
LIN {X -0.152,Y -598.274,Z 1415.130,A 0.000,B 0.000,C 90.000,E1 59.410} C_DIS
LIN {X 0.176,Y -599.975,Z 1415.120,A 0.000,B 0.000,C 90.000,E1 57.533} C_DIS
LIN {X -0.033,Y -600.950,Z 1415.114,A 0.000,B 0.000,C 90.000,E1 56.501} C_DIS
LIN {X -0.318,Y -602.609,Z 1415.104,A 0.000,B 0.000,C 90.000,E1 54.689} C_DIS
LIN {X 0.115,Y -603.705,Z 1415.096,A 0.000,B 0.000,C 90.000,E1 53.336} C_DIS
LIN {X -0.024,Y -604.866,Z 1415.088,A 0.000,B 0.000,C 90.000,E1 51.778} C_DIS
LIN {X 0.339,Y -605.777,Z 1415.080,A 0.000,B 0.000,C 90.000,E1 50.436} C_DIS
LIN {X -0.134,Y -606.344,Z 1415.073,A 0.000,B 0.000,C 90.000,E1 49.175} C_DIS
LIN {X -0.013,Y -606.530,Z 1415.067,A 0.000,B 0.000,C 90.000,E1 48.119} C_DIS
LIN {X 0.131,Y -606.753,Z 1415.059,A 0.000,B 0.000,C 90.000,E1 46.539} C_DIS
LIN {X -0.004,Y -606.769,Z 1415.054,A 0.000,B 0.000,C 90.000,E1 45.769} C_DIS
LIN {X 0.331,Y -606.590,Z 1415.047,A 0.000,B 0.000,C 90.000,E1 44.433} C_DIS
LIN {X 0.010,Y -606.221,Z 1415.041,A 0.000,B 0.000,C 90.000,E1 43.419} C_DIS
LIN {X 0.096,Y -605.673,Z 1415.036,A 0.000,B 0.000,C 90.000,E1 42.366} C_DIS
LIN {X 0.210,Y -604.990,Z 1415.030,A 0.000,B 0.000,C 90.000,E1 41.310} C_DIS
LIN {X -0.141,Y -604.119,Z 1415.024,A 0.000,B 0.000,C 90.000,E1 40.297} C_DIS
LIN {X 0.076,Y -602.483,Z 1415.015,A 0.000,B 0.000,C 90.000,E1 38.705} C_DIS
LIN {X 0.140,Y -601.103,Z 1415.009,A 0.000,B 0.000,C 90.000,E1 37.649} C_DIS
LIN {X 0.041,Y -599.964,Z 1415.005,A 0.000,B 0.000,C 90.000,E1 36.870} C_DIS
LIN {X 0.174,Y -598.185,Z 1414.999,A 0.000,B 0.000,C 90.000,E1 35.804} C_DIS
LIN {X -0.061,Y -596.051,Z 1414.993,A 0.000,B 0.000,C 90.000,E1 34.771} C_DIS
LIN {X -0.207,Y -594.307,Z 1414.989,A 0.000,B 0.000,C 90.000,E1 33.992} C_DIS
LIN {X 0.214,Y -590.967,Z 1414.981,A 0.000,B 0.000,C 90.000,E1 32.625} C_DIS
LIN {X -0.314,Y -588.680,Z 1414.977,A 0.000,B 0.000,C 90.000,E1 31.878} C_DIS
